REGION Network 3: Hardware Clock Memory 0.1S
   // 系统程序段 / System program segment
   RUNG wire#powerrail
      Contact( "Sys".COM.AlwaysON )
      wire#w1
      Contact( "ClockMemory0.1s" )
      Coil( "Sys".COM.FlashTime100mS )
   END_RUNG
   RUNG wire#w1
      Contact( "ClockMemory0.2s" )
      Coil( "Sys".COM.FlashTime200mS )
   END_RUNG
   RUNG wire#w1
      Contact( "ClockMemory0.5s" )
      Coil( "Sys".COM.FlashTime500mS )
   END_RUNG
   RUNG wire#w1
      Contact( "ClockMemory1s" )
      Coil( "Sys".COM.FlashTime1S )
   END_RUNG
   RUNG wire#w1
      Contact( "ClockMemory2s" )
      Coil( "Sys".COM.FlashTime2S )
   END_RUNG
   // the same network as SCL:
   "Sys".COM.FlashTime100mS := "Sys".COM.AlwaysON AND "ClockMemory0.1s";
   "Sys".COM.FlashTime200mS := "Sys".COM.AlwaysON AND "ClockMemory0.2s";
   "Sys".COM.FlashTime500mS := "Sys".COM.AlwaysON AND "ClockMemory0.5s";
   "Sys".COM.FlashTime1S := "Sys".COM.AlwaysON AND "ClockMemory1s";
   "Sys".COM.FlashTime2S := "Sys".COM.AlwaysON AND "ClockMemory2s";
END_REGION

REGION Network 4: Date and time config
   // 系统程序段 / System program segment
   RUNG wire#powerrail
      Contact( "Sys".DateTime.Trigger )
      { S7_Templates := "date_type := Date_And_Time" } WR_SYS_T(IN := "Sys".DateTime.Set, RET_VAL => "Sys".RETVALI)
      R_Coil( "Sys".DateTime.Trigger )
   END_RUNG
   // the same network as SCL:
   "Sys".RETVALI := WR_SYS_T(EN := "Sys".DateTime.Trigger, IN := "Sys".DateTime.Set, ENO => #_w1);
   IF #_w1 THEN "Sys".DateTime.Trigger := FALSE; END_IF;
END_REGION

REGION Network 5: Diagnostic
   RUNG wire#powerrail
      "Diagnostic"(iCPUType := 2, iDBNum := 3001, iOffset := 132, iHardwareID := "Local~PROFINET_IO-System", oStatus => "DiagnosticDataBlock".Profinet.PNReadStatus)
   END_RUNG
   // the same network as SCL:
   "Diagnostic"(iCPUType := 2,
                iDBNum := 3001,
                iOffset := 132,
                iHardwareID := "Local~PROFINET_IO-System",
                oStatus => "DiagnosticDataBlock".Profinet.PNReadStatus);
END_REGION

REGION Network 6 (SCL): Win
       "ST10_GeneralData".HMI.Win.WinBullfer := 0;
       FOR #i := 1 TO 10 DO
           "ST10_GeneralData".HMI.Win.WinBullfer := "ST10_GeneralData".HMI.Win.WinBullfer + "ST10_GeneralData".HMI.Win."10x弹窗"[#i] * 11 +"ST10_GeneralData".HMI.Win."20x弹窗"[2] * 21 +"ST10_GeneralData".HMI.Win."30x弹窗"[#i] * 31 +"ST10_GeneralData".HMI.Win."40x弹窗"[#i] * 41;
       END_FOR;
       "ST10_GeneralData".HMI.Win.WinBullfer := ABS("ST10_GeneralData".HMI.Win.WinBullfer);
       "ST10_GeneralData".HMI.Win.TON[1](IN := "ST10_GeneralData".HMI.Win.Win <> "ST10_GeneralData".HMI.Win.WinBullfer,
                          PT := T#0.5S);
   IF "ST10_GeneralData".HMI.Win.TON[1].Q THEN
       "ST10_GeneralData".HMI.Win.Win := "ST10_GeneralData".HMI.Win.WinBullfer;
       END_IF;
END_REGION

REGION Network 7: MES_Shopworx
END_REGION

REGION Network 8: Call Main
   // 系统程序段 / System program segment
   RUNG wire#powerrail
      "ST10_Main"()
   END_RUNG
   // the same network as SCL:
   "ST10_Main"();
END_REGION

REGION Network 9: DataHandling in HMI
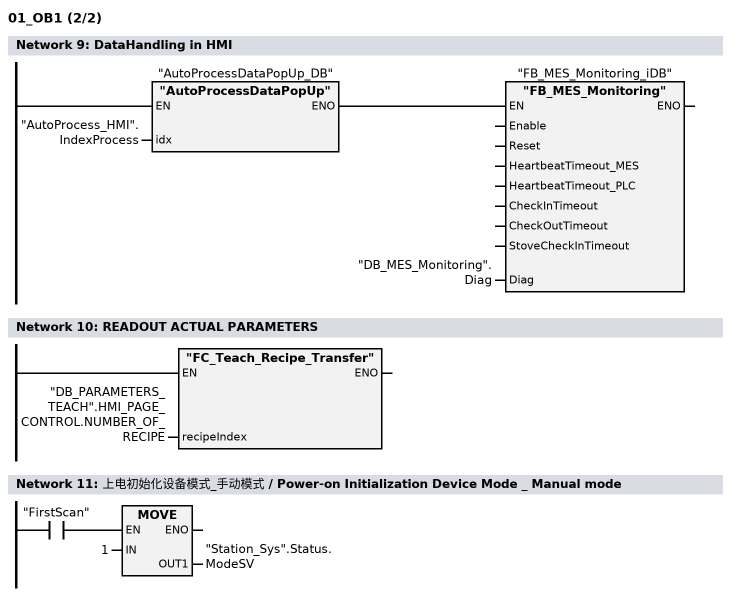
   RUNG wire#powerrail
      "AutoProcessDataPopUp_DB"(idx := "AutoProcess_HMI".IndexProcess)
      "FB_MES_Monitoring_iDB"(Enable :=, Reset :=, HeartbeatTimeout_MES :=, HeartbeatTimeout_PLC :=, CheckInTimeout :=, CheckOutTimeout :=, StoveCheckInTimeout :=, Diag := "DB_MES_Monitoring".Diag)
   END_RUNG
   // the same network as SCL:
   "AutoProcessDataPopUp_DB"(idx := "AutoProcess_HMI".IndexProcess, ENO => #_w1);   // "AutoProcessDataPopUp"
   IF #_w1 THEN
       "FB_MES_Monitoring_iDB"(Diag := "DB_MES_Monitoring".Diag);   // "FB_MES_Monitoring"
   END_IF;
END_REGION

REGION Network 10: READOUT ACTUAL PARAMETERS
   RUNG wire#powerrail
      "FC_Teach_Recipe_Transfer"(recipeIndex := "DB_PARAMETERS_TEACH".HMI_PAGE_CONTROL.NUMBER_OF_RECIPE)
   END_RUNG
   // the same network as SCL:
   "FC_Teach_Recipe_Transfer"(recipeIndex := "DB_PARAMETERS_TEACH".HMI_PAGE_CONTROL.NUMBER_OF_RECIPE);
END_REGION

REGION Network 11: 上电初始化设备模式_手动模式 / Power-on Initialization Device Mode _ Manual mode
   RUNG wire#powerrail
      Contact( "FirstScan" )
      Move(in := 1, out1 => "Station_Sys".Status.ModeSV)
   END_RUNG
   // the same network as SCL:
   IF "FirstScan" THEN "Station_Sys".Status.ModeSV := 1; END_IF;
END_REGION
END_ORGANIZATION_BLOCK

FUNCTION "Diagnostic" : Void   // FC3001, SCL
TITLE = Diagnostic
{ S7_Optimized_Access := 'FALSE' }
AUTHOR : STD
FAMILY : RCS
VERSION : 18.0
// stored: AutoNumber false, SetENOAutomatically true
   VAR_INPUT
      iCPUType : Int;   // 1-DP&PN 2-PN
      iDBNum : Word;
      iOffset : Int;   // Start address
      iHardwareID : HW_IOSYSTEM;
   END_VAR
   VAR_OUTPUT
      oStatus : Int;
   END_VAR
   VAR_TEMP
      RDSRet : Struct
         Busy : Bool;
         Header : Struct
            Length : Word;
            Number : Word;
         END_STRUCT;
      END_STRUCT;
      retInt : Int;
      SSL : Struct
         SSID : Word;
         Index : Word;
         Length : Int;
      END_STRUCT;
      DR : Any;
      DRS AT DR : Struct
         SyntaxID : Byte;
         DataType : Byte;
         RepetitionFactor : Int;
         DB_Number : Word;
         MemoryAreaAddress : DWord;
      END_STRUCT;
   END_VAR
BEGIN

   (*############################################################
      RUHLAMAT SUZHOU ELEC.STD.
      Copyright (c) 2017. All rights reserved.    

      NAME OF FUNCTION BLOCK:         Diagnostic
      VERSION NUMBER:                 V3.0
      COMPOSER:                       Ming.Jiang

      CreateDate:                    16.Nov.2016
      ----------------------------------------------------------
      Interface description:
      IN:
          "iCPUType"
          iDBNum
          iOffset
          iHardwareID

      INOUT:
      OUT:
          oStatus

      ----------------------------------------------------------
      #RET_VALUE:

      #Alert Value:

      ----------------------------------------------------------
      Date           Name      Version           Activity                                                                              
      28.Nov.2016    JM        V3.0              add alarm

   ############################################################*)
   IF #iCPUType = 0 OR #iDBNum = 0 THEN
       ENO := 0;
       RETURN;
   ELSE
       IF #iCPUType=2 THEN
           GOTO PN;
       ELSIF #iCPUType=1 THEN
           ;
       ELSE
           ENO := 0;
           RETURN;
       END_IF;
       #DRS.SyntaxID := 16#10;
       #DRS.DataType := 16#02;
       #DRS.RepetitionFactor := 128;
       #DRS.DB_Number := #iDBNum;
       #DRS.MemoryAreaAddress := 16#8400_0000 OR (SHL(IN := INT_TO_DWORD(#iOffset), N := 3));
       #oStatus := DeviceStates(LADDR := #iHardwareID, MODE := 2, STATE := #DR);
   PN:
       #DRS.SyntaxID := 16#10;
       #DRS.DataType := 16#02;
       #DRS.RepetitionFactor := 128;
       #DRS.DB_Number := #iDBNum;
       #DRS.MemoryAreaAddress := 16#8400_0000 OR (SHL(IN := INT_TO_DWORD(#iOffset), N := 3));
       #oStatus := DeviceStates(LADDR := #iHardwareID, MODE := 2, STATE := #DR);
       // orginise interface data 
       ENO := 1;
       RETURN;
   END_IF;
END_FUNCTION

FUNCTION "ST10_Main" : Void   // FC1050, LAD
{ S7_Optimized_Access := 'FALSE' }
// //=====================================================
// // INFO
// //=====================================================
// // NAME : ST10_Main
// // EN   : Main control logic for OP010 station.
// // ZH   : OP010 主控制逻辑。
// // SK   : Hlavná riadiaca logika stanice OP010.
// //=====================================================
// stored: AutoNumber false, SetENOAutomatically false
BEGIN

REGION Network 1 (SCL): INFO
   //=====================================================
   // INFO
   //=====================================================
   // NAME : ST10_Main
   // EN   : Main control logic for OP010 station.
   // ZH   : OP010 主控制逻辑。
   // SK   : Hlavná riadiaca logika stanice OP010.
   //=====================================================
END_REGION

REGION Network 2
   // 系统功能组调用部分
   // 1.该部分用户可以自己根据系统的组成将需要的功能块调用写在该部分
   // 2.该部分禁止与系统功能无关的程序在此处调用
END_REGION

NETWORK
TITLE = XXXX=====Station Relation/工位相关 =====StartXXXXX / XXXX=====Station Relation/Station correlation =====StartXXXXX

REGION Network 4: input /输入
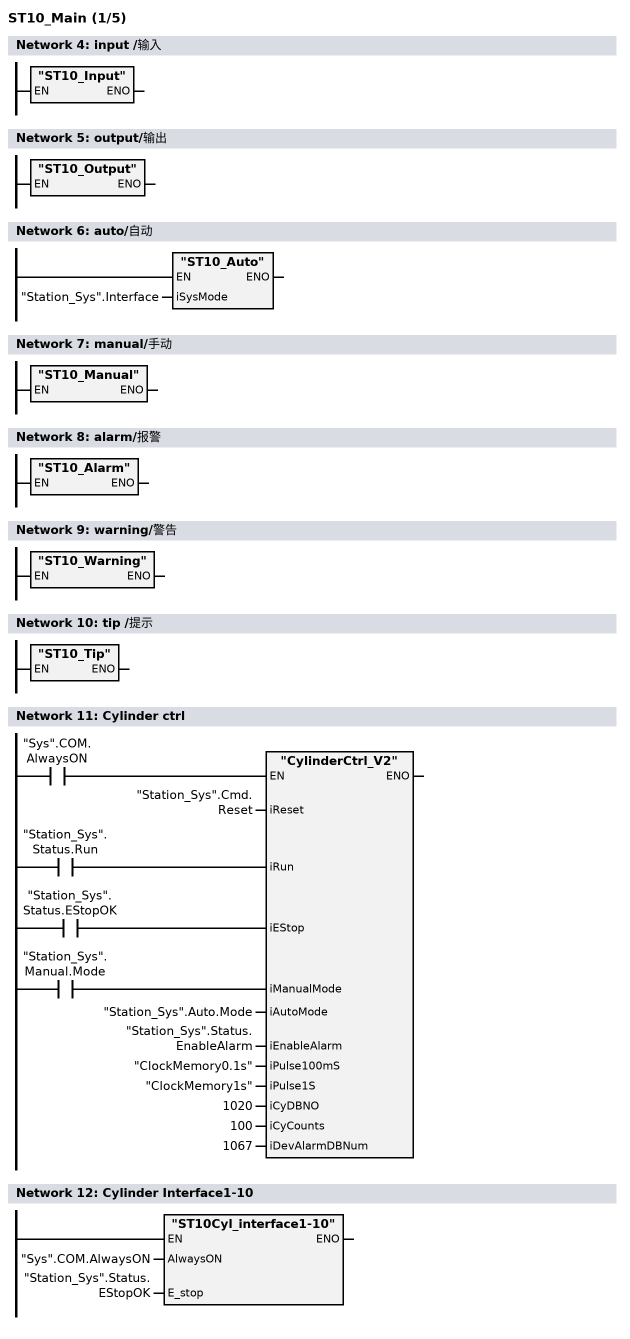
   RUNG wire#powerrail
      "ST10_Input"()
   END_RUNG
   // the same network as SCL:
   "ST10_Input"();
END_REGION

REGION Network 5: output/输出
   RUNG wire#powerrail
      "ST10_Output"()
   END_RUNG
   // the same network as SCL:
   "ST10_Output"();
END_REGION

REGION Network 6: auto/自动
   RUNG wire#powerrail
      "ST10_Auto"(iSysMode := "Station_Sys".Interface)
   END_RUNG
   // the same network as SCL:
   "ST10_Auto"(iSysMode := "Station_Sys".Interface);
END_REGION

REGION Network 7: manual/手动
   RUNG wire#powerrail
      "ST10_Manual"()
   END_RUNG
   // the same network as SCL:
   "ST10_Manual"();
END_REGION

REGION Network 8: alarm/报警
   RUNG wire#powerrail
      "ST10_Alarm"()
   END_RUNG
   // the same network as SCL:
   "ST10_Alarm"();
END_REGION

REGION Network 9: warning/警告
   RUNG wire#powerrail
      "ST10_Warning"()
   END_RUNG
   // the same network as SCL:
   "ST10_Warning"();
END_REGION

REGION Network 10: tip /提示
   RUNG wire#powerrail
      "ST10_Tip"()
   END_RUNG
   // the same network as SCL:
   "ST10_Tip"();
END_REGION

REGION Network 11: Cylinder ctrl
   RUNG wire#powerrail
      Contact( "Sys".COM.AlwaysON )
      "CylinderCtrl_V2"(iRun := wire#w1, iEStop := wire#w2, iManualMode := wire#w3, iReset := "Station_Sys".Cmd.Reset, iAutoMode := "Station_Sys".Auto.Mode, iEnableAlarm := "Station_Sys".Status.EnableAlarm, iPulse100mS := "ClockMemory0.1s", iPulse1S := "ClockMemory1s", iCyDBNO := 1020, iCyCounts := 100, iDevAlarmDBNum := 1067)
   END_RUNG
   RUNG wire#powerrail
      Contact( "Station_Sys".Status.Run )
   END_RUNG wire#w1
   RUNG wire#powerrail
      Contact( "Station_Sys".Status.EStopOK )
   END_RUNG wire#w2
   RUNG wire#powerrail
      Contact( "Station_Sys".Manual.Mode )
   END_RUNG wire#w3
   // the same network as SCL:
   IF "Sys".COM.AlwaysON THEN
       "CylinderCtrl_V2"(iReset := "Station_Sys".Cmd.Reset,
                         iRun := "Station_Sys".Status.Run,
                         iEStop := "Station_Sys".Status.EStopOK,
                         iManualMode := "Station_Sys".Manual.Mode,
                         iAutoMode := "Station_Sys".Auto.Mode,
                         iEnableAlarm := "Station_Sys".Status.EnableAlarm,
                         iPulse100mS := "ClockMemory0.1s",
                         iPulse1S := "ClockMemory1s",
                         iCyDBNO := 1020,
                         iCyCounts := 100,
                         iDevAlarmDBNum := 1067);
   END_IF;
END_REGION

REGION Network 12: Cylinder Interface1-10
   RUNG wire#powerrail
      "ST10Cyl_interface1-10"(AlwaysON := "Sys".COM.AlwaysON, E_stop := "Station_Sys".Status.EStopOK)
   END_RUNG
   // the same network as SCL:
   "ST10Cyl_interface1-10"(AlwaysON := "Sys".COM.AlwaysON, E_stop := "Station_Sys".Status.EStopOK);
END_REGION

REGION Network 13: Cylinder Interface11-20
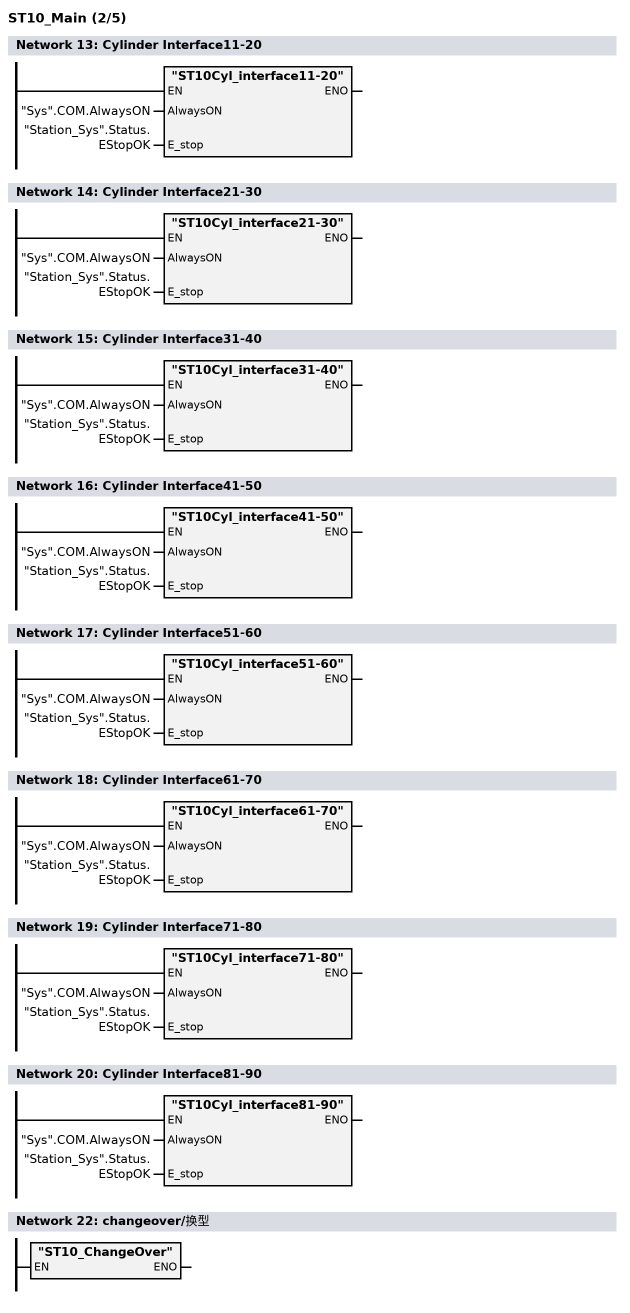
   RUNG wire#powerrail
      "ST10Cyl_interface11-20"(AlwaysON := "Sys".COM.AlwaysON, E_stop := "Station_Sys".Status.EStopOK)
   END_RUNG
   // the same network as SCL:
   "ST10Cyl_interface11-20"(AlwaysON := "Sys".COM.AlwaysON, E_stop := "Station_Sys".Status.EStopOK);
END_REGION

REGION Network 14: Cylinder Interface21-30
   RUNG wire#powerrail
      "ST10Cyl_interface21-30"(AlwaysON := "Sys".COM.AlwaysON, E_stop := "Station_Sys".Status.EStopOK)
   END_RUNG
   // the same network as SCL:
   "ST10Cyl_interface21-30"(AlwaysON := "Sys".COM.AlwaysON, E_stop := "Station_Sys".Status.EStopOK);
END_REGION

REGION Network 15: Cylinder Interface31-40
   RUNG wire#powerrail
      "ST10Cyl_interface31-40"(AlwaysON := "Sys".COM.AlwaysON, E_stop := "Station_Sys".Status.EStopOK)
   END_RUNG
   // the same network as SCL:
   "ST10Cyl_interface31-40"(AlwaysON := "Sys".COM.AlwaysON, E_stop := "Station_Sys".Status.EStopOK);
END_REGION

REGION Network 16: Cylinder Interface41-50
   RUNG wire#powerrail
      "ST10Cyl_interface41-50"(AlwaysON := "Sys".COM.AlwaysON, E_stop := "Station_Sys".Status.EStopOK)
   END_RUNG
   // the same network as SCL:
   "ST10Cyl_interface41-50"(AlwaysON := "Sys".COM.AlwaysON, E_stop := "Station_Sys".Status.EStopOK);
END_REGION

REGION Network 17: Cylinder Interface51-60
   RUNG wire#powerrail
      "ST10Cyl_interface51-60"(AlwaysON := "Sys".COM.AlwaysON, E_stop := "Station_Sys".Status.EStopOK)
   END_RUNG
   // the same network as SCL:
   "ST10Cyl_interface51-60"(AlwaysON := "Sys".COM.AlwaysON, E_stop := "Station_Sys".Status.EStopOK);
END_REGION

REGION Network 18: Cylinder Interface61-70
   RUNG wire#powerrail
      "ST10Cyl_interface61-70"(AlwaysON := "Sys".COM.AlwaysON, E_stop := "Station_Sys".Status.EStopOK)
   END_RUNG
   // the same network as SCL:
   "ST10Cyl_interface61-70"(AlwaysON := "Sys".COM.AlwaysON, E_stop := "Station_Sys".Status.EStopOK);
END_REGION

REGION Network 19: Cylinder Interface71-80
   RUNG wire#powerrail
      "ST10Cyl_interface71-80"(AlwaysON := "Sys".COM.AlwaysON, E_stop := "Station_Sys".Status.EStopOK)
   END_RUNG
   // the same network as SCL:
   "ST10Cyl_interface71-80"(AlwaysON := "Sys".COM.AlwaysON, E_stop := "Station_Sys".Status.EStopOK);
END_REGION

REGION Network 20: Cylinder Interface81-90
   RUNG wire#powerrail
      "ST10Cyl_interface81-90"(AlwaysON := "Sys".COM.AlwaysON, E_stop := "Station_Sys".Status.EStopOK)
   END_RUNG
   // the same network as SCL:
   "ST10Cyl_interface81-90"(AlwaysON := "Sys".COM.AlwaysON, E_stop := "Station_Sys".Status.EStopOK);
END_REGION

REGION Network 22: changeover/换型
   RUNG wire#powerrail
      "ST10_ChangeOver"()
   END_RUNG
   // the same network as SCL:
   "ST10_ChangeOver"();
END_REGION

REGION Network 23: Device
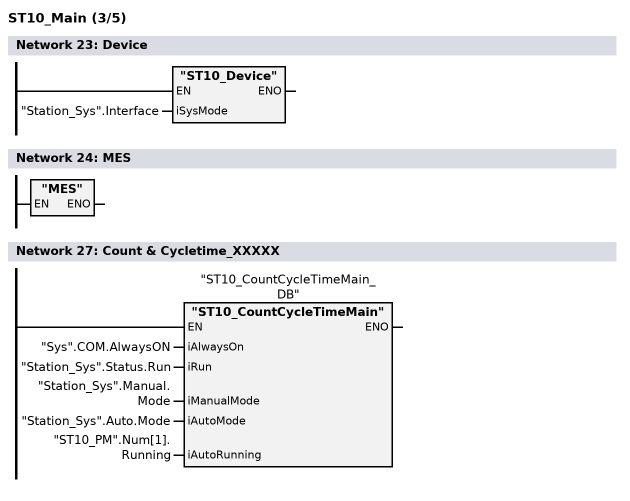
   RUNG wire#powerrail
      "ST10_Device"(iSysMode := "Station_Sys".Interface)
   END_RUNG
   // the same network as SCL:
   "ST10_Device"(iSysMode := "Station_Sys".Interface);
END_REGION

REGION Network 24: MES
   RUNG wire#powerrail
      "MES"()
   END_RUNG
   // the same network as SCL:
   "MES"();
END_REGION

REGION Network 25: =====System Function related information Section =====Start
END_REGION

NETWORK
TITLE = SystemFunction IO

REGION Network 27: Count & Cycletime_XXXXX
   RUNG wire#powerrail
      "ST10_CountCycleTimeMain_DB"(iAlwaysOn := "Sys".COM.AlwaysON, iRun := "Station_Sys".Status.Run, iManualMode := "Station_Sys".Manual.Mode, iAutoMode := "Station_Sys".Auto.Mode, iAutoRunning := "ST10_PM".Num[1].Running)
   END_RUNG
   // the same network as SCL:
   "ST10_CountCycleTimeMain_DB"(iAlwaysOn := "Sys".COM.AlwaysON,   // "ST10_CountCycleTimeMain"
                           iRun := "Station_Sys".Status.Run,
                           iManualMode := "Station_Sys".Manual.Mode,
                           iAutoMode := "Station_Sys".Auto.Mode,
                           iAutoRunning := "ST10_PM".Num[1].Running);
END_REGION

REGION Network 28: System mode
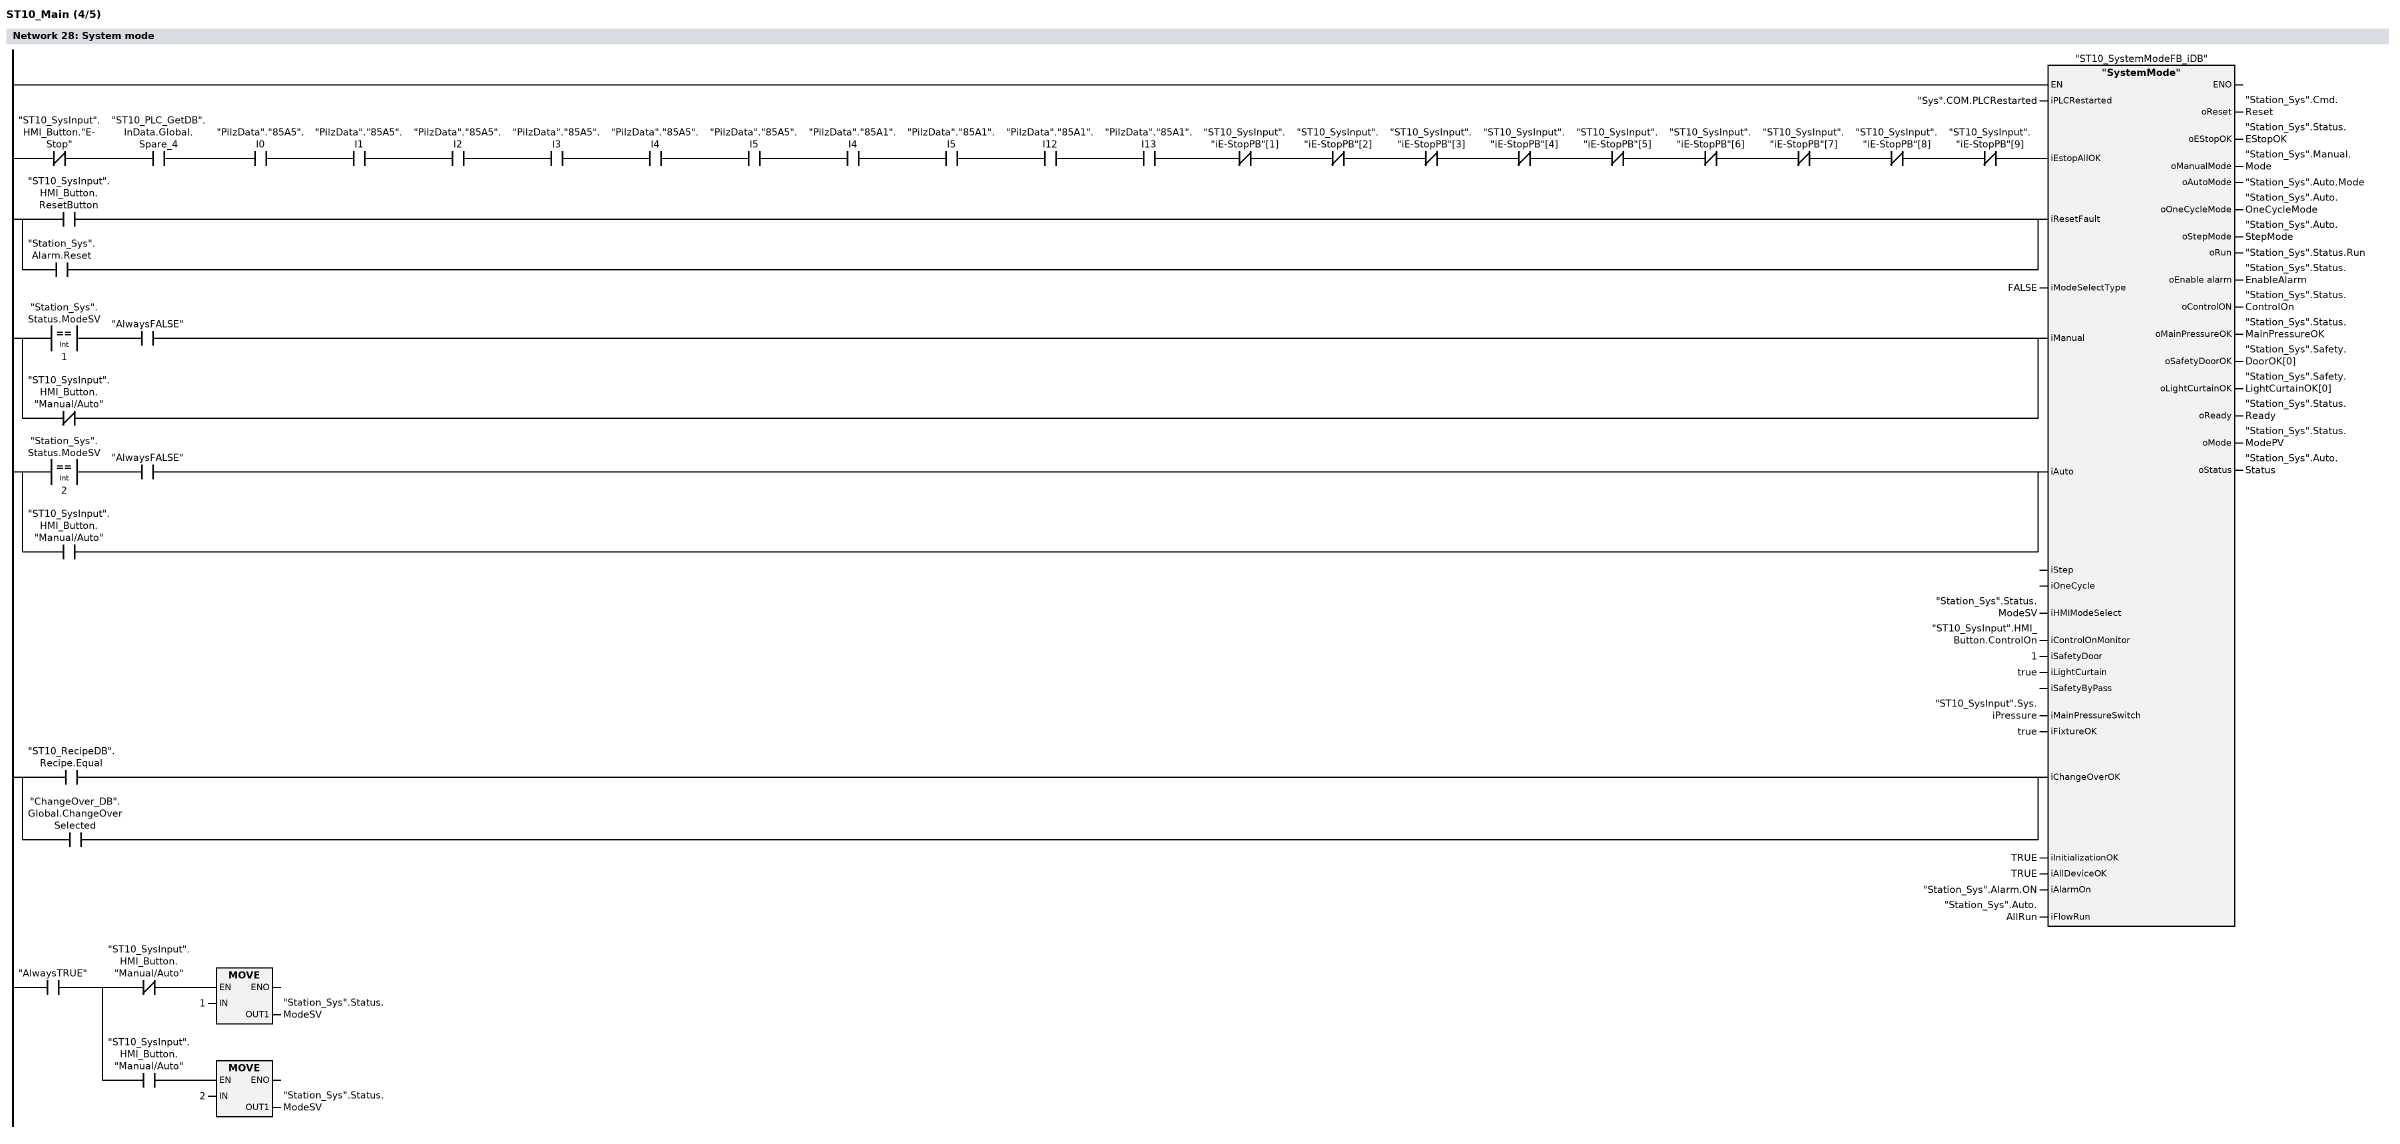
   RUNG wire#powerrail
      "ST10_SystemModeFB_iDB"(iEstopAllOK := wire#w1, iResetFault := wire#w2, iManual := wire#w3, iAuto := wire#w4, iChangeOverOK := wire#w5, iPLCRestarted := "Sys".COM.PLCRestarted, iModeSelectType := FALSE, iStep :=, iOneCycle :=, iHMIModeSelect := "Station_Sys".Status.ModeSV, iControlOnMonitor := "ST10_SysInput".HMI_Button.ControlOn, iSafetyDoor := 1, iLightCurtain := true, iSafetyByPass :=, iMainPressureSwitch := "ST10_SysInput".Sys.iPressure, iFixtureOK := true, iInitializationOK := TRUE, iAllDeviceOK := TRUE, iAlarmOn := "Station_Sys".Alarm.ON, iFlowRun := "Station_Sys".Auto.AllRun, oReset => "Station_Sys".Cmd.Reset, oEStopOK => "Station_Sys".Status.EStopOK, oManualMode => "Station_Sys".Manual.Mode, oAutoMode => "Station_Sys".Auto.Mode, oOneCycleMode => "Station_Sys".Auto.OneCycleMode, oStepMode => "Station_Sys".Auto.StepMode, oRun => "Station_Sys".Status.Run, "oEnable alarm" => "Station_Sys".Status.EnableAlarm, oControlON => "Station_Sys".Status.ControlOn, oMainPressureOK => "Station_Sys".Status.MainPressureOK, oSafetyDoorOK => "Station_Sys".Safety.DoorOK[0], oLightCurtainOK => "Station_Sys".Safety.LightCurtainOK[0], oReady => "Station_Sys".Status.Ready, oMode => "Station_Sys".Status.ModePV, oStatus => "Station_Sys".Auto.Status)
   END_RUNG
   RUNG wire#powerrail
      I_Contact( "ST10_SysInput".HMI_Button."E-Stop" )
      Contact( "ST10_PLC_GetDB".InData.Global.Spare_4 )
      Contact( "PilzData"."85A5".I0 )
      Contact( "PilzData"."85A5".I1 )
      Contact( "PilzData"."85A5".I2 )
      Contact( "PilzData"."85A5".I3 )
      Contact( "PilzData"."85A5".I4 )
      Contact( "PilzData"."85A5".I5 )
      Contact( "PilzData"."85A1".I4 )
      Contact( "PilzData"."85A1".I5 )
      Contact( "PilzData"."85A1".I12 )
      Contact( "PilzData"."85A1".I13 )
      I_Contact( "ST10_SysInput"."iE-StopPB"[1] )
      I_Contact( "ST10_SysInput"."iE-StopPB"[2] )
      I_Contact( "ST10_SysInput"."iE-StopPB"[3] )
      I_Contact( "ST10_SysInput"."iE-StopPB"[4] )
      I_Contact( "ST10_SysInput"."iE-StopPB"[5] )
      I_Contact( "ST10_SysInput"."iE-StopPB"[6] )
      I_Contact( "ST10_SysInput"."iE-StopPB"[7] )
      I_Contact( "ST10_SysInput"."iE-StopPB"[8] )
      I_Contact( "ST10_SysInput"."iE-StopPB"[9] )
   END_RUNG wire#w1
   RUNG wire#powerrail
      Contact( "ST10_SysInput".HMI_Button.ResetButton )
   END_RUNG wire#w2
   RUNG wire#powerrail
      Contact( "Station_Sys".Alarm.Reset )
   END_RUNG wire#w2
   RUNG wire#powerrail
      { S7_Templates := "SrcType := Int" } EQ_Contact(in1 := "Station_Sys".Status.ModeSV, in2 := 1)
      Contact( "AlwaysFALSE" )
   END_RUNG wire#w3
   RUNG wire#powerrail
      I_Contact( "ST10_SysInput".HMI_Button."Manual/Auto" )
   END_RUNG wire#w3
   RUNG wire#powerrail
      { S7_Templates := "SrcType := Int" } EQ_Contact(in1 := "Station_Sys".Status.ModeSV, in2 := 2)
      Contact( "AlwaysFALSE" )
   END_RUNG wire#w4
   RUNG wire#powerrail
      Contact( "ST10_SysInput".HMI_Button."Manual/Auto" )
   END_RUNG wire#w4
   RUNG wire#powerrail
      Contact( "ST10_RecipeDB".Recipe.Equal )
   END_RUNG wire#w5
   RUNG wire#powerrail
      Contact( "ChangeOver_DB".Global.ChangeOverSelected )
   END_RUNG wire#w5
   RUNG wire#powerrail
      Contact( "AlwaysTRUE" )
      wire#w6
      I_Contact( "ST10_SysInput".HMI_Button."Manual/Auto" )
      Move(in := 1, out1 => "Station_Sys".Status.ModeSV)
   END_RUNG
   RUNG wire#w6
      Contact( "ST10_SysInput".HMI_Button."Manual/Auto" )
      Move(in := 2, out1 => "Station_Sys".Status.ModeSV)
   END_RUNG
   // the same network as SCL:
   "ST10_SystemModeFB_iDB"(iPLCRestarted := "Sys".COM.PLCRestarted,   // "SystemMode"
                           iEstopAllOK := NOT "ST10_SysInput".HMI_Button."E-Stop" AND "ST10_PLC_GetDB".InData.Global.Spare_4 AND "PilzData"."85A5".I0 AND "PilzData"."85A5".I1 AND "PilzData"."85A5".I2 AND "PilzData"."85A5".I3 AND "PilzData"."85A5".I4 AND "PilzData"."85A5".I5 AND "PilzData"."85A1".I4 AND "PilzData"."85A1".I5 AND "PilzData"."85A1".I12 AND "PilzData"."85A1".I13 AND NOT "ST10_SysInput"."iE-StopPB"[1] AND NOT "ST10_SysInput"."iE-StopPB"[2] AND NOT "ST10_SysInput"."iE-StopPB"[3] AND NOT "ST10_SysInput"."iE-StopPB"[4] AND NOT "ST10_SysInput"."iE-StopPB"[5] AND NOT "ST10_SysInput"."iE-StopPB"[6] AND NOT "ST10_SysInput"."iE-StopPB"[7] AND NOT "ST10_SysInput"."iE-StopPB"[8] AND NOT "ST10_SysInput"."iE-StopPB"[9],
                           iResetFault := "ST10_SysInput".HMI_Button.ResetButton OR "Station_Sys".Alarm.Reset,
                           iModeSelectType := FALSE,
                           iManual := (("Station_Sys".Status.ModeSV = 1) AND "AlwaysFALSE") OR NOT "ST10_SysInput".HMI_Button."Manual/Auto",
                           iAuto := (("Station_Sys".Status.ModeSV = 2) AND "AlwaysFALSE") OR "ST10_SysInput".HMI_Button."Manual/Auto",
                           iHMIModeSelect := "Station_Sys".Status.ModeSV,
                           iControlOnMonitor := "ST10_SysInput".HMI_Button.ControlOn,
                           iSafetyDoor := 1,
                           iLightCurtain := true,
                           iMainPressureSwitch := "ST10_SysInput".Sys.iPressure,
                           iFixtureOK := true,
                           iChangeOverOK := "ST10_RecipeDB".Recipe.Equal OR "ChangeOver_DB".Global.ChangeOverSelected,
                           iInitializationOK := TRUE,
                           iAllDeviceOK := TRUE,
                           iAlarmOn := "Station_Sys".Alarm.ON,
                           iFlowRun := "Station_Sys".Auto.AllRun,
                           oReset => "Station_Sys".Cmd.Reset,
                           oEStopOK => "Station_Sys".Status.EStopOK,
                           oManualMode => "Station_Sys".Manual.Mode,
                           oAutoMode => "Station_Sys".Auto.Mode,
                           oOneCycleMode => "Station_Sys".Auto.OneCycleMode,
                           oStepMode => "Station_Sys".Auto.StepMode,
                           oRun => "Station_Sys".Status.Run,
                           "oEnable alarm" => "Station_Sys".Status.EnableAlarm,
                           oControlON => "Station_Sys".Status.ControlOn,
                           oMainPressureOK => "Station_Sys".Status.MainPressureOK,
                           oSafetyDoorOK => "Station_Sys".Safety.DoorOK[0],
                           oLightCurtainOK => "Station_Sys".Safety.LightCurtainOK[0],
                           oReady => "Station_Sys".Status.Ready,
                           oMode => "Station_Sys".Status.ModePV,
                           oStatus => "Station_Sys".Auto.Status);
   IF "AlwaysTRUE" AND NOT "ST10_SysInput".HMI_Button."Manual/Auto" THEN
       "Station_Sys".Status.ModeSV := 1;
   END_IF;
   IF "AlwaysTRUE" AND "ST10_SysInput".HMI_Button."Manual/Auto" THEN
       "Station_Sys".Status.ModeSV := 2;
   END_IF;
END_REGION

REGION Network 29: Start button
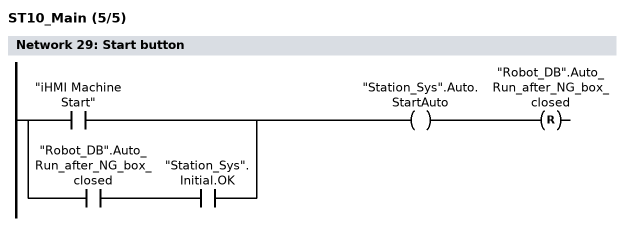
   RUNG wire#powerrail
      Contact( "iHMI Machine Start" )
      wire#w1
      Coil( "Station_Sys".Auto.StartAuto )
      R_Coil( "Robot_DB".Auto_Run_after_NG_box_closed )
   END_RUNG
   RUNG wire#powerrail
      Contact( "Robot_DB".Auto_Run_after_NG_box_closed )
      Contact( "Station_Sys".Initial.OK )
   END_RUNG wire#w1
   // the same network as SCL:
   "Station_Sys".Auto.StartAuto := "iHMI Machine Start" OR ("Robot_DB".Auto_Run_after_NG_box_closed AND "Station_Sys".Initial.OK);
   IF "Station_Sys".Auto.StartAuto THEN "Robot_DB".Auto_Run_after_NG_box_closed := FALSE; END_IF;
END_REGION

REGION Network 30 (SCL): System Interface
   "Station_Sys".Interface.CPUFristCycle  := "Sys".COM.PLCRestarted;
   "Station_Sys".Interface.SysRun         := "Station_Sys".Status.Run;
   "Station_Sys".Interface.Reset          := "Station_Sys".Cmd.Reset;
   "Station_Sys".Interface.EstopOK        := "Station_Sys".Status.EStopOK;
   "Station_Sys".Interface.SafetyDoorOK   := "Station_Sys".Safety.DoorOK[0];
   "Station_Sys".Interface.LightCurtainOK := "Station_Sys".Safety.LightCurtainOK[0];
   "Station_Sys".Interface.SetInitial     := "Station_Sys".Initial.Set;
   "Station_Sys".Interface.InitialRun     := "Station_Sys".Initial.Running;
   "Station_Sys".Interface.Ready          := "Station_Sys".Status.Ready;
   "Station_Sys".Interface.ManualMode     := "Station_Sys".Manual.Mode;
   "Station_Sys".Interface.Auto           := "Station_Sys".Auto;
END_REGION

REGION Network 31: =====System Function related information Section =====End
END_REGION

REGION Network 32: CallCalibration//标定调用
END_REGION

REGION Network 33 (SCL): ByPass Button
   // A
   "ST10_GeneralData".FunctionDeSelect.A.FunctionDeSelected_Servo380A1  := "ST10_GeneralData".FunctionDeSelect.A.DeSelectPB_Servo380A1;
   "ST10_GeneralData".FunctionDeSelect.A.FunctionDeSelected_Servo381A1  := "ST10_GeneralData".FunctionDeSelect.A.DeSelectPB_Servo381A1;
   "ST10_GeneralData".FunctionDeSelect.A.FunctionDeSelected_Servo383A1  := "ST10_GeneralData".FunctionDeSelect.A.DeSelectPB_Servo383A1;
   "ST10_GeneralData".FunctionDeSelect.A.FunctionDeSelected_Reader800A1 := "ST10_GeneralData".FunctionDeSelect.A.DeSelectPB_Reader800A1;
   "ST10_GeneralData".FunctionDeSelect.A.FunctionDeSelected_Reader801A1 := "ST10_GeneralData".FunctionDeSelect.A.DeSelectPB_Reader801A1;
   "ST10_GeneralData".FunctionDeSelect.A.FunctionDeSelected_Reader802A1 := "ST10_GeneralData".FunctionDeSelect.A.DeSelectPB_Reader802A1;
   "ST10_GeneralData".FunctionDeSelect.A.FunctionDeSelected_Reader803A1 := "ST10_GeneralData".FunctionDeSelect.A.DeSelectPB_Reader803A1;
   "ST10_GeneralData".FunctionDeSelect.A.FunctionDeSelected_Reader804A1 := "ST10_GeneralData".FunctionDeSelect.A.DeSelectPB_Reader804A1;

   // B
   "ST10_GeneralData".FunctionDeSelect.B.FunctionDeSelected_Press372A1     := "ST10_GeneralData".FunctionDeSelect.B.DeSelectPB_Press372A1;
   "ST10_GeneralData".FunctionDeSelect.B.FunctionDeSelected_Press375A1     := "ST10_GeneralData".FunctionDeSelect.B.DeSelectPB_Press375A1;
   "ST10_GeneralData".FunctionDeSelect.B.FunctionDeSelected_Reader806A1    := "ST10_GeneralData".FunctionDeSelect.B.DeSelectPB_Reader806A1;
   "ST10_GeneralData".FunctionDeSelect.B.FunctionDeSelected_TestPress372A1 := "ST10_GeneralData".FunctionDeSelect.B.DeSelectPB_TestPress372A1;
   "ST10_GeneralData".FunctionDeSelect.B.FunctionDeSelected_TestPress375A1 := "ST10_GeneralData".FunctionDeSelect.B.DeSelectPB_TestPress375A1;

   // C
   "ST10_GeneralData".FunctionDeSelect.C.FunctionDeSelected_Servo382A1 := "ST10_GeneralData".FunctionDeSelect.C.DeSelectPB_Servo382A1;
   "ST10_GeneralData".FunctionDeSelect.C.FunctionDeSelected_ServoIAI := "ST10_GeneralData".FunctionDeSelect.C.DeSelectPB_ServoIAI;
   "ST10_GeneralData".FunctionDeSelect.C.FunctionDeSelected_IV3810A1 := "ST10_GeneralData".FunctionDeSelect.C.DeSelectPB_IV3810A1;
   "ST10_GeneralData".FunctionDeSelect.C.FunctionDeSelected_IV3811A1 := "ST10_GeneralData".FunctionDeSelect.C.DeSelectPB_IV3811A1;
   "ST10_GeneralData".FunctionDeSelect.C.FunctionDeSelected_Glue := "ST10_GeneralData".FunctionDeSelect.C.DeSelectPB_Glue;

   // E
   "ST10_GeneralData".FunctionDeSelect.E.FunctionDeSelected := "ST10_GeneralData".FunctionDeSelect.E.DeSelectPB;

   // F
   "ST10_GeneralData".FunctionDeSelect.F.FunctionDeSelected_Reader805A1 := "ST10_GeneralData".FunctionDeSelect.F.DeSelectPB_Reader805A1;

   // H
   "ST10_GeneralData".FunctionDeSelect.H.FunctionDeSelected := "ST10_GeneralData".FunctionDeSelect.H.DeSelectPB;

   // J
   "ST10_GeneralData".FunctionDeSelect.J.FunctionDeSelected := "ST10_GeneralData".FunctionDeSelect.J.DeSelectPB;

   // K
   "ST10_GeneralData".FunctionDeSelect.K.FunctionDeSelected := "ST10_GeneralData".FunctionDeSelect.K.DeSelectPB;

   // L
   "ST10_GeneralData".FunctionDeSelect.L.FunctionDeSelected := "ST10_GeneralData".FunctionDeSelect.L.DeSelectPB;

   // MES
   "ST10_GeneralData".FunctionDeSelect.MES.FunctionDeSelected := "ST10_GeneralData".FunctionDeSelect.MES.DeSelectPB;

   //Auto>Maanual  ScanFixture
   "ST10_GeneralData".FunctionDeSelect.Global.FunctionDeSelected_ScanFixture := "ST10_GeneralData".FunctionDeSelect.Global.DeSelectPB_ScanFixture;
END_REGION
END_FUNCTION

FUNCTION "ST10_Input" : Void   // FC1001, LAD
{ S7_Optimized_Access := 'FALSE' }
VERSION : 0.1
// 注：本程序用来处理需要滤波，延时、计算的输入信号
// stored: AutoNumber false, IsIECCheckEnabled false, SetENOAutomatically false, UDAEnableTagReadback false
BEGIN

REGION Network 1 (SCL): HMI信号映射 / HMI signal mapping
   "ST10_SysInput".HMI_Button.ControlOn := "iHMI Control On";
   //"ST350_SysInput".HMI_Button.ControlOff:=
   "ST10_SysInput".HMI_Button.MachineStart := "iHMI Machine Start";
   "ST10_SysInput".HMI_Button.MachineStop := "iHMI Machine Stop";
   "ST10_SysInput".HMI_Button.ResetButton := "iHMI ResetButton";
   "ST10_SysInput".HMI_Button."Manual/Auto" := "iHMI Manual/Auto";
   "ST10_SysInput".HMI_Button.SafetyGateUnlock := "iHMI Safety Gate Unlock";
   "ST10_SysInput".HMI_Button."E-Stop" :=  "iHMI E-Stop";
END_REGION

REGION Network 2 (SCL): Sys IO Image
   "ST10_SysInput".Sys.iCircuitBreakerOK1 := "iCircuit Breaker OK_1";
   "ST10_SysInput".Sys.iCircuitBreakerOK2 := "iCircuit Breaker OK_2";
   "ST10_SysInput".Sys.iPressure:= "iPressure";
END_REGION

REGION Network 3 (SCL): iE-StopPB
   "ST10_SysInput"."iE-StopPB"[1] := "iE_StopButton2_A01";
   "ST10_SysInput"."iE-StopPB"[2] := "iE_StopButton3_A02";
   "ST10_SysInput"."iE-StopPB"[3] := "iE_StopButton4_H";
   "ST10_SysInput"."iE-StopPB"[4] := "iE_StopButton5_J";
   "ST10_SysInput"."iE-StopPB"[5] := "iE_StopButton6_K";
   "ST10_SysInput"."iE-StopPB"[6] := "iE_StopButton7_L";
   "ST10_SysInput"."iE-StopPB"[7] := "iH_StopButton";
   "ST10_SysInput"."iE-StopPB"[8] := "iJ_StopButton";
   "ST10_SysInput"."iE-StopPB"[9] := "iK_StopButton";
END_REGION

REGION Network 4 (SCL): iSafetyGatFeedBack
   (*
   "ST350_SysInput".iSafetyGatFeedBack[1] := "iSafety door Locking FeedBack_1";
   "ST350_SysInput".iSafetyGatFeedBack[2] := "iSafety door Locking FeedBack_2";
   "ST350_SysInput".iSafetyGatFeedBack[3] := "iSafety door Locking FeedBack_3";
   "ST350_SysInput".iSafetyGatFeedBack[4] := "iSafety door Locking FeedBack_4";
   "ST350_SysInput".iSafetyGatFeedBack[5] := "iSafety door Locking FeedBack_5";
   "ST350_SysInput".iSafetyGatFeedBack[6] := "iSafety door Locking FeedBack_6";
   "ST350_SysInput".iSafetyGatFeedBack[7] := "iSafety door Locking FeedBack_7";
   "ST350_SysInput".iSafetyGatFeedBack[8] := "iSafety door Locking FeedBack_8";
   *)
END_REGION

REGION Network 5 (SCL): iSafetydoorLockingFeedBack
   "ST10_SysInput".iSafetydoorLockingFeedBack[1] := "iSafety door Locking FeedBack_1";
   "ST10_SysInput".iSafetydoorLockingFeedBack[2] := "iSafety door Locking FeedBack_2";
   "ST10_SysInput".iSafetydoorLockingFeedBack[3] := "iSafety door Locking FeedBack_3";
   "ST10_SysInput".iSafetydoorLockingFeedBack[4] := "iSafety door Locking FeedBack_4";
   "ST10_SysInput".iSafetydoorLockingFeedBack[5] := "iSafety door Locking FeedBack_5";
   "ST10_SysInput".iSafetydoorLockingFeedBack[6] := "iSafety door Locking FeedBack_6";
   "ST10_SysInput".iSafetydoorLockingFeedBack[7] := "iSafety door Locking FeedBack_7";
   "ST10_SysInput".iSafetydoorLockingFeedBack[8] := "iSafety door Locking FeedBack_8";
END_REGION

REGION Network 6 (SCL): iSafetydoorLockingFeedBack
   "ST10_SysInput".iMaterieldoorLockingFeedBack[1] := "iMateriel Door Locking FeedBack_H1";
   "ST10_SysInput".iMaterieldoorLockingFeedBack[2] := "iMateriel Door Locking FeedBack_H2";
   "ST10_SysInput".iMaterieldoorLockingFeedBack[3] := "iMateriel Door Locking FeedBack_J1";
   "ST10_SysInput".iMaterieldoorLockingFeedBack[4] := "iMateriel Door Locking FeedBack_J2";
   "ST10_SysInput".iMaterieldoorLockingFeedBack[5] := "iMateriel Door Locking FeedBack_K1";
   "ST10_SysInput".iMaterieldoorLockingFeedBack[6] := "iMateriel Door Locking FeedBack_K2";
   "ST10_SysInput".iMaterieldoorLockingFeedBack[7] := "iMateriel Door Locking FeedBack_L1";
END_REGION
END_FUNCTION

FUNCTION "ST10_Output" : Void   // FC1002, LAD
{ S7_Optimized_Access := 'FALSE' }
// stored: AutoNumber false, SetENOAutomatically false
   VAR_TEMP   // added for the SCL form of the ladder/FBD networks
      _w1 : Bool;
      _w2 : Bool;
      _w3 : Bool;
      _w4 : Bool;
      _w5 : Bool;
      _w6 : Bool;
   END_VAR
BEGIN

REGION Network 1 (SCL): 安全门锁定信号映射SafetyDoorCoil / Security door lock_1
   "oSafetyDoorLocked_1" := "ST10_SysOutput".SafetyDoorCoil[1];
   "oSafetyDoorLocked_2" := "ST10_SysOutput".SafetyDoorCoil[2];
   "oSafetyDoorLocked_3" := "ST10_SysOutput".SafetyDoorCoil[3];
   "oSafetyDoorLocked_4" := "ST10_SysOutput".SafetyDoorCoil[4];
   "oSafetyDoorLocked_5" := "ST10_SysOutput".SafetyDoorCoil[5];
   "oSafetyDoorLocked_6" := "ST10_SysOutput".SafetyDoorCoil[6];
   "oSafetyDoorLocked_7" := "ST10_SysOutput".SafetyDoorCoil[7];
   "oSafetyDoorLocked_8" := "ST10_SysOutput".SafetyDoorCoil[8];
   "oSafetyDoorLocked" := "ST10_SysOutput".SafetyDoorCoil[9];
END_REGION

REGION Network 2 (SCL): 安全门锁定信号映射SafetyDoorCoil / Material door lock_1
   "oMaterielDoorLocked_H1" := "ST10_SysOutput".MaterialDoorCoil[1];
   "oMaterielDoorLocked_H2" := "ST10_SysOutput".MaterialDoorCoil[2];
   "oMaterielDoorLocked_J1" := "ST10_SysOutput".MaterialDoorCoil[3];
   "oMaterielDoorLocked_J2" := "ST10_SysOutput".MaterialDoorCoil[4];
   "oMaterielDoorLocked_K1" := "ST10_SysOutput".MaterialDoorCoil[5];
   "oMaterielDoorLocked_K2" := "ST10_SysOutput".MaterialDoorCoil[6];
   "oMaterielDoorLocked_L1" := "ST10_SysOutput".MaterialDoorCoil[7];


   "oE-NG-01SafetyGate" := "ST10_SysOutput".MaterialDoorCoil[8];
   "oE-NG-02SafetyGate" := "ST10_SysOutput".MaterialDoorCoil[9];
END_REGION

REGION Network 3: 塔灯
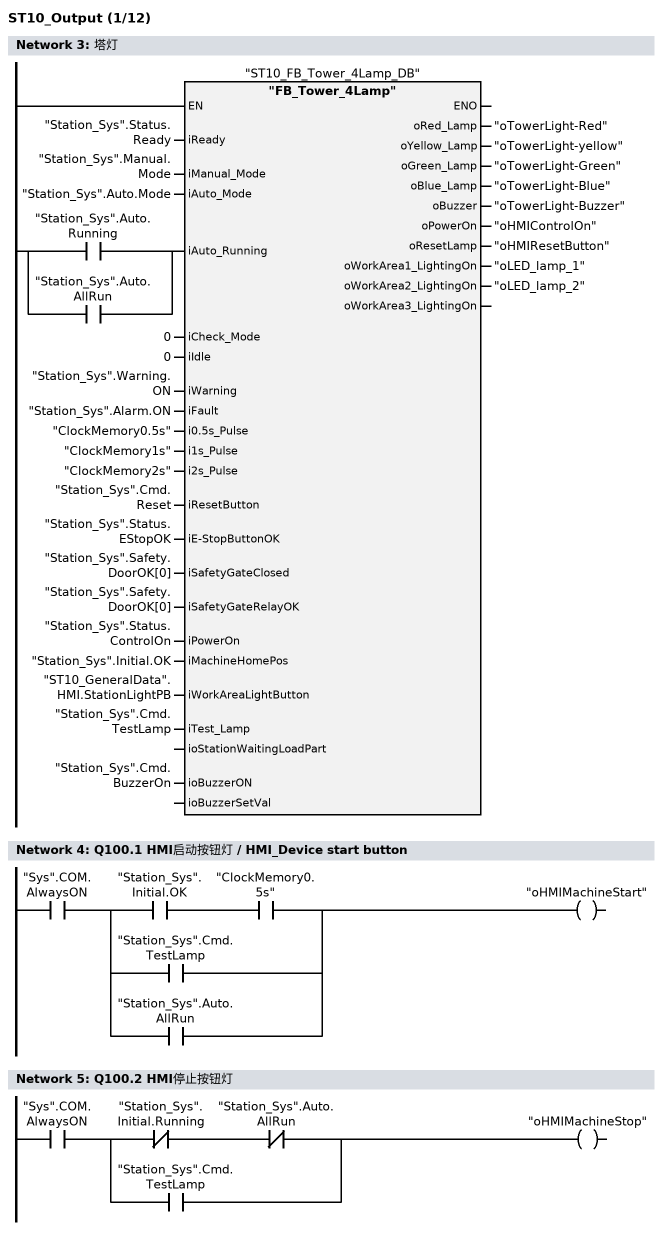
   RUNG wire#powerrail
      "ST10_FB_Tower_4Lamp_DB"(iAuto_Running := wire#w1, iReady := "Station_Sys".Status.Ready, iManual_Mode := "Station_Sys".Manual.Mode, iAuto_Mode := "Station_Sys".Auto.Mode, iCheck_Mode := 0, iIdle := 0, iWarning := "Station_Sys".Warning.ON, iFault := "Station_Sys".Alarm.ON, "i0.5s_Pulse" := "ClockMemory0.5s", i1s_Pulse := "ClockMemory1s", i2s_Pulse := "ClockMemory2s", iResetButton := "Station_Sys".Cmd.Reset, "iE-StopButtonOK" := "Station_Sys".Status.EStopOK, iSafetyGateClosed := "Station_Sys".Safety.DoorOK[0], iSafetyGateRelayOK := "Station_Sys".Safety.DoorOK[0], iPowerOn := "Station_Sys".Status.ControlOn, iMachineHomePos := "Station_Sys".Initial.OK, iWorkAreaLightButton := "ST10_GeneralData".HMI.StationLightPB, iTest_Lamp := "Station_Sys".Cmd.TestLamp, ioStationWaitingLoadPart :=, ioBuzzerON := "Station_Sys".Cmd.BuzzerOn, ioBuzzerSetVal :=, oRed_Lamp => "oTowerLight-Red", oYellow_Lamp => "oTowerLight-yellow", oGreen_Lamp => "oTowerLight-Green", oBlue_Lamp => "oTowerLight-Blue", oBuzzer => "oTowerLight-Buzzer", oPowerOn => "oHMIControlOn", oResetLamp => "oHMIResetButton", oWorkArea1_LightingOn => "oLED_lamp_1", oWorkArea2_LightingOn => "oLED_lamp_2", oWorkArea3_LightingOn =>)
   END_RUNG
   RUNG wire#powerrail
      Contact( "Station_Sys".Auto.Running )
   END_RUNG wire#w1
   RUNG wire#powerrail
      Contact( "Station_Sys".Auto.AllRun )
   END_RUNG wire#w1
   // the same network as SCL:
   "ST10_FB_Tower_4Lamp_DB"(iReady := "Station_Sys".Status.Ready,   // "FB_Tower_4Lamp"
                           iManual_Mode := "Station_Sys".Manual.Mode,
                           iAuto_Mode := "Station_Sys".Auto.Mode,
                           iAuto_Running := "Station_Sys".Auto.Running OR "Station_Sys".Auto.AllRun,
                           iCheck_Mode := 0,
                           iIdle := 0,
                           iWarning := "Station_Sys".Warning.ON,
                           iFault := "Station_Sys".Alarm.ON,
                           "i0.5s_Pulse" := "ClockMemory0.5s",
                           i1s_Pulse := "ClockMemory1s",
                           i2s_Pulse := "ClockMemory2s",
                           iResetButton := "Station_Sys".Cmd.Reset,
                           "iE-StopButtonOK" := "Station_Sys".Status.EStopOK,
                           iSafetyGateClosed := "Station_Sys".Safety.DoorOK[0],
                           iSafetyGateRelayOK := "Station_Sys".Safety.DoorOK[0],
                           iPowerOn := "Station_Sys".Status.ControlOn,
                           iMachineHomePos := "Station_Sys".Initial.OK,
                           iWorkAreaLightButton := "ST10_GeneralData".HMI.StationLightPB,
                           iTest_Lamp := "Station_Sys".Cmd.TestLamp,
                           ioBuzzerON := "Station_Sys".Cmd.BuzzerOn,
                           oRed_Lamp => "oTowerLight-Red",
                           oYellow_Lamp => "oTowerLight-yellow",
                           oGreen_Lamp => "oTowerLight-Green",
                           oBlue_Lamp => "oTowerLight-Blue",
                           oBuzzer => "oTowerLight-Buzzer",
                           oPowerOn => "oHMIControlOn",
                           oResetLamp => "oHMIResetButton",
                           oWorkArea1_LightingOn => "oLED_lamp_1",
                           oWorkArea2_LightingOn => "oLED_lamp_2");
END_REGION

REGION Network 4: Q100.1 HMI启动按钮灯 / HMI_Device start button
   RUNG wire#powerrail
      Contact( "Sys".COM.AlwaysON )
      wire#w1
      Contact( "Station_Sys".Initial.OK )
      Contact( "ClockMemory0.5s" )
      wire#w2
      Coil( "oHMIMachineStart" )
   END_RUNG
   RUNG wire#w1
      Contact( "Station_Sys".Cmd.TestLamp )
   END_RUNG wire#w2
   RUNG wire#w1
      Contact( "Station_Sys".Auto.AllRun )
   END_RUNG wire#w2
   // the same network as SCL:
   "oHMIMachineStart" := "Sys".COM.AlwaysON AND (("Station_Sys".Initial.OK AND "ClockMemory0.5s") OR "Station_Sys".Cmd.TestLamp OR "Station_Sys".Auto.AllRun);
END_REGION

REGION Network 5: Q100.2 HMI停止按钮灯
   RUNG wire#powerrail
      Contact( "Sys".COM.AlwaysON )
      wire#w1
      I_Contact( "Station_Sys".Initial.Running )
      I_Contact( "Station_Sys".Auto.AllRun )
      wire#w2
      Coil( "oHMIMachineStop" )
   END_RUNG
   RUNG wire#w1
      Contact( "Station_Sys".Cmd.TestLamp )
   END_RUNG wire#w2
   // the same network as SCL:
   "oHMIMachineStop" := "Sys".COM.AlwaysON AND ((NOT "Station_Sys".Initial.Running AND NOT "Station_Sys".Auto.AllRun) OR "Station_Sys".Cmd.TestLamp);
END_REGION

REGION Network 6: Q100.4 HMI开门按钮灯
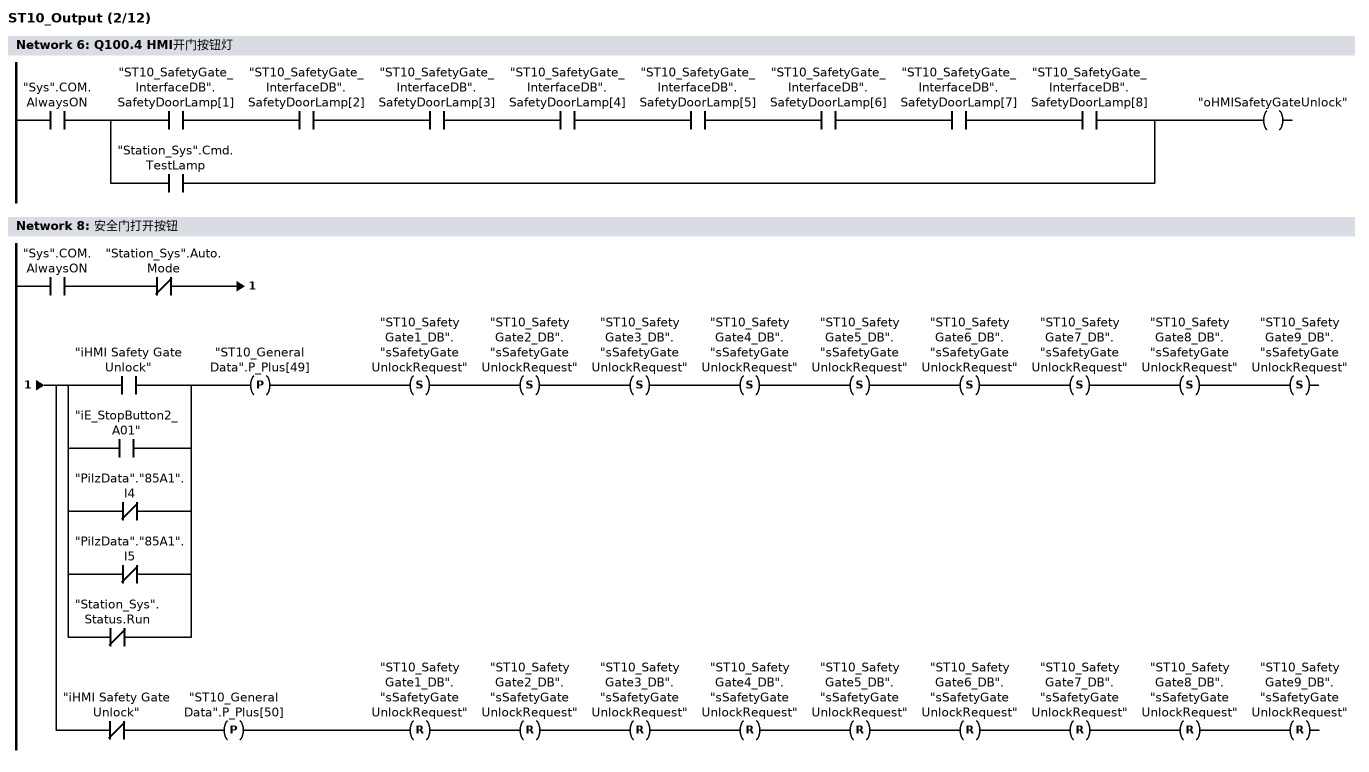
   RUNG wire#powerrail
      Contact( "Sys".COM.AlwaysON )
      wire#w1
      Contact( "ST10_SafetyGate_InterfaceDB".SafetyDoorLamp[1] )
      Contact( "ST10_SafetyGate_InterfaceDB".SafetyDoorLamp[2] )
      Contact( "ST10_SafetyGate_InterfaceDB".SafetyDoorLamp[3] )
      Contact( "ST10_SafetyGate_InterfaceDB".SafetyDoorLamp[4] )
      Contact( "ST10_SafetyGate_InterfaceDB".SafetyDoorLamp[5] )
      Contact( "ST10_SafetyGate_InterfaceDB".SafetyDoorLamp[6] )
      Contact( "ST10_SafetyGate_InterfaceDB".SafetyDoorLamp[7] )
      Contact( "ST10_SafetyGate_InterfaceDB".SafetyDoorLamp[8] )
      wire#w2
      Coil( "oHMISafetyGateUnlock" )
   END_RUNG
   RUNG wire#w1
      Contact( "Station_Sys".Cmd.TestLamp )
   END_RUNG wire#w2
   // the same network as SCL:
   "oHMISafetyGateUnlock" := "Sys".COM.AlwaysON AND (("ST10_SafetyGate_InterfaceDB".SafetyDoorLamp[1] AND "ST10_SafetyGate_InterfaceDB".SafetyDoorLamp[2] AND "ST10_SafetyGate_InterfaceDB".SafetyDoorLamp[3] AND "ST10_SafetyGate_InterfaceDB".SafetyDoorLamp[4] AND "ST10_SafetyGate_InterfaceDB".SafetyDoorLamp[5] AND "ST10_SafetyGate_InterfaceDB".SafetyDoorLamp[6] AND "ST10_SafetyGate_InterfaceDB".SafetyDoorLamp[7] AND "ST10_SafetyGate_InterfaceDB".SafetyDoorLamp[8]) OR "Station_Sys".Cmd.TestLamp);
END_REGION

REGION Network 8: 安全门打开按钮
   RUNG wire#powerrail
      Contact( "Sys".COM.AlwaysON )
      I_Contact( "Station_Sys".Auto.Mode )
      wire#w1
      Contact( "iHMI Safety Gate Unlock" )
      wire#w2
      P_Trig( "ST10_GeneralData".P_Plus[49] )
      S_Coil( "ST10_SafetyGate1_DB"."sSafetyGate UnlockRequest" )
      S_Coil( "ST10_SafetyGate2_DB"."sSafetyGate UnlockRequest" )
      S_Coil( "ST10_SafetyGate3_DB"."sSafetyGate UnlockRequest" )
      S_Coil( "ST10_SafetyGate4_DB"."sSafetyGate UnlockRequest" )
      S_Coil( "ST10_SafetyGate5_DB"."sSafetyGate UnlockRequest" )
      S_Coil( "ST10_SafetyGate6_DB"."sSafetyGate UnlockRequest" )
      S_Coil( "ST10_SafetyGate7_DB"."sSafetyGate UnlockRequest" )
      S_Coil( "ST10_SafetyGate8_DB"."sSafetyGate UnlockRequest" )
      S_Coil( "ST10_SafetyGate9_DB"."sSafetyGate UnlockRequest" )
   END_RUNG
   RUNG wire#w1
      Contact( "iE_StopButton2_A01" )
   END_RUNG wire#w2
   RUNG wire#w1
      I_Contact( "PilzData"."85A1".I4 )
   END_RUNG wire#w2
   RUNG wire#w1
      I_Contact( "PilzData"."85A1".I5 )
   END_RUNG wire#w2
   RUNG wire#w1
      I_Contact( "Station_Sys".Status.Run )
   END_RUNG wire#w2
   RUNG wire#w1
      I_Contact( "iHMI Safety Gate Unlock" )
      P_Trig( "ST10_GeneralData".P_Plus[50] )
      R_Coil( "ST10_SafetyGate1_DB"."sSafetyGate UnlockRequest" )
      R_Coil( "ST10_SafetyGate2_DB"."sSafetyGate UnlockRequest" )
      R_Coil( "ST10_SafetyGate3_DB"."sSafetyGate UnlockRequest" )
      R_Coil( "ST10_SafetyGate4_DB"."sSafetyGate UnlockRequest" )
      R_Coil( "ST10_SafetyGate5_DB"."sSafetyGate UnlockRequest" )
      R_Coil( "ST10_SafetyGate6_DB"."sSafetyGate UnlockRequest" )
      R_Coil( "ST10_SafetyGate7_DB"."sSafetyGate UnlockRequest" )
      R_Coil( "ST10_SafetyGate8_DB"."sSafetyGate UnlockRequest" )
      R_Coil( "ST10_SafetyGate9_DB"."sSafetyGate UnlockRequest" )
   END_RUNG
   // the same network as SCL:
   #_w1 := "Sys".COM.AlwaysON AND NOT "Station_Sys".Auto.Mode;
   #_w2 := #_w1 AND ("iHMI Safety Gate Unlock" OR "iE_StopButton2_A01" OR NOT "PilzData"."85A1".I4 OR NOT "PilzData"."85A1".I5 OR NOT "Station_Sys".Status.Run);
   #_w3 := #_w2 AND NOT "ST10_GeneralData".P_Plus[49];   // rising edge
   "ST10_GeneralData".P_Plus[49] := #_w2;
   IF #_w3 THEN
       "ST10_SafetyGate1_DB"."sSafetyGate UnlockRequest" := TRUE;
       "ST10_SafetyGate2_DB"."sSafetyGate UnlockRequest" := TRUE;
       "ST10_SafetyGate3_DB"."sSafetyGate UnlockRequest" := TRUE;
       "ST10_SafetyGate4_DB"."sSafetyGate UnlockRequest" := TRUE;
       "ST10_SafetyGate5_DB"."sSafetyGate UnlockRequest" := TRUE;
       "ST10_SafetyGate6_DB"."sSafetyGate UnlockRequest" := TRUE;
       "ST10_SafetyGate7_DB"."sSafetyGate UnlockRequest" := TRUE;
       "ST10_SafetyGate8_DB"."sSafetyGate UnlockRequest" := TRUE;
       "ST10_SafetyGate9_DB"."sSafetyGate UnlockRequest" := TRUE;
   END_IF;
   #_w4 := #_w1 AND NOT "iHMI Safety Gate Unlock";
   #_w5 := #_w4 AND NOT "ST10_GeneralData".P_Plus[50];   // rising edge
   "ST10_GeneralData".P_Plus[50] := #_w4;
   IF #_w5 THEN
       "ST10_SafetyGate1_DB"."sSafetyGate UnlockRequest" := FALSE;
       "ST10_SafetyGate2_DB"."sSafetyGate UnlockRequest" := FALSE;
       "ST10_SafetyGate3_DB"."sSafetyGate UnlockRequest" := FALSE;
       "ST10_SafetyGate4_DB"."sSafetyGate UnlockRequest" := FALSE;
       "ST10_SafetyGate5_DB"."sSafetyGate UnlockRequest" := FALSE;
       "ST10_SafetyGate6_DB"."sSafetyGate UnlockRequest" := FALSE;
       "ST10_SafetyGate7_DB"."sSafetyGate UnlockRequest" := FALSE;
       "ST10_SafetyGate8_DB"."sSafetyGate UnlockRequest" := FALSE;
       "ST10_SafetyGate9_DB"."sSafetyGate UnlockRequest" := FALSE;
   END_IF;
END_REGION

REGION Network 9: 安全门关闭
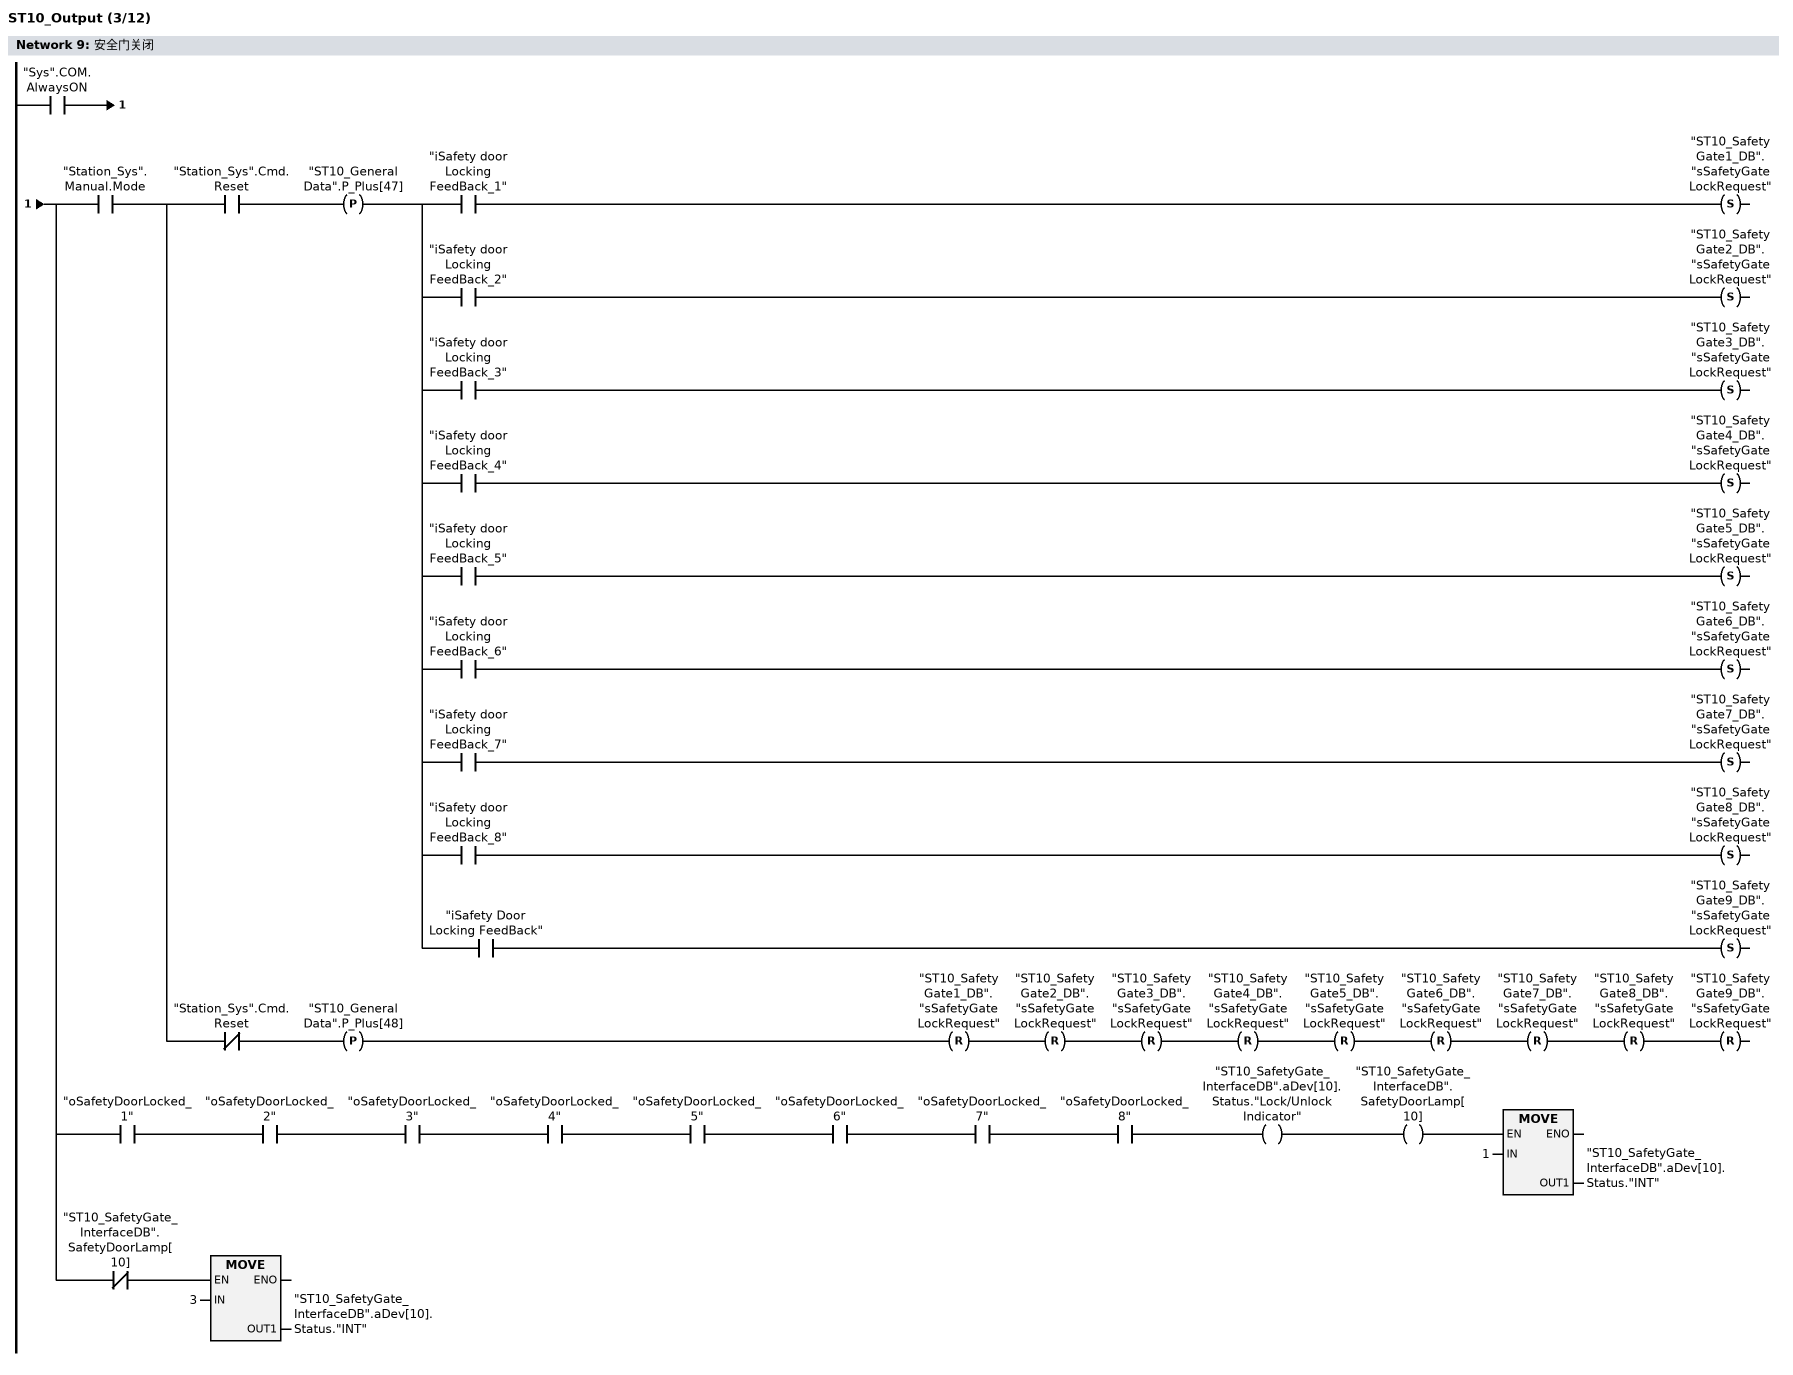
   RUNG wire#powerrail
      Contact( "Sys".COM.AlwaysON )
      wire#w1
      Contact( "Station_Sys".Manual.Mode )
      wire#w2
      Contact( "Station_Sys".Cmd.Reset )
      P_Trig( "ST10_GeneralData".P_Plus[47] )
      wire#w3
      Contact( "iSafety door Locking FeedBack_1" )
      S_Coil( "ST10_SafetyGate1_DB"."sSafetyGate LockRequest" )
   END_RUNG
   RUNG wire#w3
      Contact( "iSafety door Locking FeedBack_2" )
      S_Coil( "ST10_SafetyGate2_DB"."sSafetyGate LockRequest" )
   END_RUNG
   RUNG wire#w3
      Contact( "iSafety door Locking FeedBack_3" )
      S_Coil( "ST10_SafetyGate3_DB"."sSafetyGate LockRequest" )
   END_RUNG
   RUNG wire#w3
      Contact( "iSafety door Locking FeedBack_4" )
      S_Coil( "ST10_SafetyGate4_DB"."sSafetyGate LockRequest" )
   END_RUNG
   RUNG wire#w3
      Contact( "iSafety door Locking FeedBack_5" )
      S_Coil( "ST10_SafetyGate5_DB"."sSafetyGate LockRequest" )
   END_RUNG
   RUNG wire#w3
      Contact( "iSafety door Locking FeedBack_6" )
      S_Coil( "ST10_SafetyGate6_DB"."sSafetyGate LockRequest" )
   END_RUNG
   RUNG wire#w3
      Contact( "iSafety door Locking FeedBack_7" )
      S_Coil( "ST10_SafetyGate7_DB"."sSafetyGate LockRequest" )
   END_RUNG
   RUNG wire#w3
      Contact( "iSafety door Locking FeedBack_8" )
      S_Coil( "ST10_SafetyGate8_DB"."sSafetyGate LockRequest" )
   END_RUNG
   RUNG wire#w3
      Contact( "iSafety Door Locking FeedBack" )
      S_Coil( "ST10_SafetyGate9_DB"."sSafetyGate LockRequest" )
   END_RUNG
   RUNG wire#w2
      I_Contact( "Station_Sys".Cmd.Reset )
      P_Trig( "ST10_GeneralData".P_Plus[48] )
      R_Coil( "ST10_SafetyGate1_DB"."sSafetyGate LockRequest" )
      R_Coil( "ST10_SafetyGate2_DB"."sSafetyGate LockRequest" )
      R_Coil( "ST10_SafetyGate3_DB"."sSafetyGate LockRequest" )
      R_Coil( "ST10_SafetyGate4_DB"."sSafetyGate LockRequest" )
      R_Coil( "ST10_SafetyGate5_DB"."sSafetyGate LockRequest" )
      R_Coil( "ST10_SafetyGate6_DB"."sSafetyGate LockRequest" )
      R_Coil( "ST10_SafetyGate7_DB"."sSafetyGate LockRequest" )
      R_Coil( "ST10_SafetyGate8_DB"."sSafetyGate LockRequest" )
      R_Coil( "ST10_SafetyGate9_DB"."sSafetyGate LockRequest" )
   END_RUNG
   RUNG wire#w1
      Contact( "oSafetyDoorLocked_1" )
      Contact( "oSafetyDoorLocked_2" )
      Contact( "oSafetyDoorLocked_3" )
      Contact( "oSafetyDoorLocked_4" )
      Contact( "oSafetyDoorLocked_5" )
      Contact( "oSafetyDoorLocked_6" )
      Contact( "oSafetyDoorLocked_7" )
      Contact( "oSafetyDoorLocked_8" )
      Coil( "ST10_SafetyGate_InterfaceDB".aDev[10].Status."Lock/Unlock Indicator" )
      Coil( "ST10_SafetyGate_InterfaceDB".SafetyDoorLamp[10] )
      Move(in := 1, out1 => "ST10_SafetyGate_InterfaceDB".aDev[10].Status."INT")
   END_RUNG
   RUNG wire#w1
      I_Contact( "ST10_SafetyGate_InterfaceDB".SafetyDoorLamp[10] )
      Move(in := 3, out1 => "ST10_SafetyGate_InterfaceDB".aDev[10].Status."INT")
   END_RUNG
   // the same network as SCL:
   #_w1 := "Sys".COM.AlwaysON AND "Station_Sys".Manual.Mode;
   #_w2 := #_w1 AND "Station_Sys".Cmd.Reset;
   #_w3 := #_w2 AND NOT "ST10_GeneralData".P_Plus[47];   // rising edge
   "ST10_GeneralData".P_Plus[47] := #_w2;
   IF #_w3 AND "iSafety door Locking FeedBack_1" THEN
       "ST10_SafetyGate1_DB"."sSafetyGate LockRequest" := TRUE;
   END_IF;
   IF #_w3 AND "iSafety door Locking FeedBack_2" THEN
       "ST10_SafetyGate2_DB"."sSafetyGate LockRequest" := TRUE;
   END_IF;
   IF #_w3 AND "iSafety door Locking FeedBack_3" THEN
       "ST10_SafetyGate3_DB"."sSafetyGate LockRequest" := TRUE;
   END_IF;
   IF #_w3 AND "iSafety door Locking FeedBack_4" THEN
       "ST10_SafetyGate4_DB"."sSafetyGate LockRequest" := TRUE;
   END_IF;
   IF #_w3 AND "iSafety door Locking FeedBack_5" THEN
       "ST10_SafetyGate5_DB"."sSafetyGate LockRequest" := TRUE;
   END_IF;
   IF #_w3 AND "iSafety door Locking FeedBack_6" THEN
       "ST10_SafetyGate6_DB"."sSafetyGate LockRequest" := TRUE;
   END_IF;
   IF #_w3 AND "iSafety door Locking FeedBack_7" THEN
       "ST10_SafetyGate7_DB"."sSafetyGate LockRequest" := TRUE;
   END_IF;
   IF #_w3 AND "iSafety door Locking FeedBack_8" THEN
       "ST10_SafetyGate8_DB"."sSafetyGate LockRequest" := TRUE;
   END_IF;
   IF #_w3 AND "iSafety Door Locking FeedBack" THEN
       "ST10_SafetyGate9_DB"."sSafetyGate LockRequest" := TRUE;
   END_IF;
   #_w4 := #_w1 AND NOT "Station_Sys".Cmd.Reset;
   #_w5 := #_w4 AND NOT "ST10_GeneralData".P_Plus[48];   // rising edge
   "ST10_GeneralData".P_Plus[48] := #_w4;
   IF #_w5 THEN
       "ST10_SafetyGate1_DB"."sSafetyGate LockRequest" := FALSE;
       "ST10_SafetyGate2_DB"."sSafetyGate LockRequest" := FALSE;
       "ST10_SafetyGate3_DB"."sSafetyGate LockRequest" := FALSE;
       "ST10_SafetyGate4_DB"."sSafetyGate LockRequest" := FALSE;
       "ST10_SafetyGate5_DB"."sSafetyGate LockRequest" := FALSE;
       "ST10_SafetyGate6_DB"."sSafetyGate LockRequest" := FALSE;
       "ST10_SafetyGate7_DB"."sSafetyGate LockRequest" := FALSE;
       "ST10_SafetyGate8_DB"."sSafetyGate LockRequest" := FALSE;
       "ST10_SafetyGate9_DB"."sSafetyGate LockRequest" := FALSE;
   END_IF;
   "ST10_SafetyGate_InterfaceDB".aDev[10].Status."Lock/Unlock Indicator" := "Sys".COM.AlwaysON AND "oSafetyDoorLocked_1" AND "oSafetyDoorLocked_2" AND "oSafetyDoorLocked_3" AND "oSafetyDoorLocked_4" AND "oSafetyDoorLocked_5" AND "oSafetyDoorLocked_6" AND "oSafetyDoorLocked_7" AND "oSafetyDoorLocked_8";
   "ST10_SafetyGate_InterfaceDB".SafetyDoorLamp[10] := "Sys".COM.AlwaysON AND "oSafetyDoorLocked_1" AND "oSafetyDoorLocked_2" AND "oSafetyDoorLocked_3" AND "oSafetyDoorLocked_4" AND "oSafetyDoorLocked_5" AND "oSafetyDoorLocked_6" AND "oSafetyDoorLocked_7" AND "oSafetyDoorLocked_8";
   IF "Sys".COM.AlwaysON AND "oSafetyDoorLocked_1" AND "oSafetyDoorLocked_2" AND "oSafetyDoorLocked_3" AND "oSafetyDoorLocked_4" AND "oSafetyDoorLocked_5" AND "oSafetyDoorLocked_6" AND "oSafetyDoorLocked_7" AND "oSafetyDoorLocked_8" THEN
       "ST10_SafetyGate_InterfaceDB".aDev[10].Status."INT" := 1;
   END_IF;
   IF "Sys".COM.AlwaysON AND NOT "ST10_SafetyGate_InterfaceDB".SafetyDoorLamp[10] THEN
       "ST10_SafetyGate_InterfaceDB".aDev[10].Status."INT" := 3;
   END_IF;
END_REGION

REGION Network 11: E-NG料盒-02安全门锁按钮灯
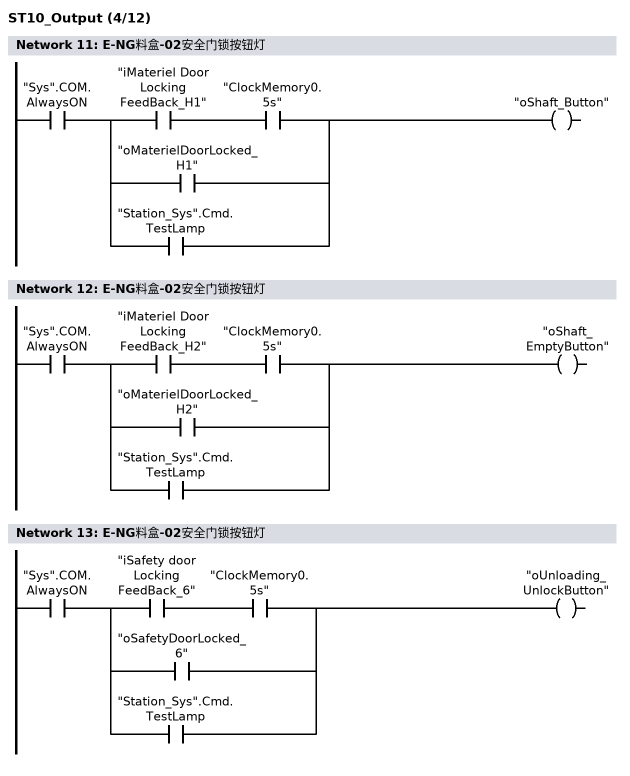
   RUNG wire#powerrail
      Contact( "Sys".COM.AlwaysON )
      wire#w1
      Contact( "iMateriel Door Locking FeedBack_H1" )
      Contact( "ClockMemory0.5s" )
      wire#w2
      Coil( "oShaft_Button" )
   END_RUNG
   RUNG wire#w1
      Contact( "oMaterielDoorLocked_H1" )
   END_RUNG wire#w2
   RUNG wire#w1
      Contact( "Station_Sys".Cmd.TestLamp )
   END_RUNG wire#w2
   // the same network as SCL:
   "oShaft_Button" := "Sys".COM.AlwaysON AND (("iMateriel Door Locking FeedBack_H1" AND "ClockMemory0.5s") OR "oMaterielDoorLocked_H1" OR "Station_Sys".Cmd.TestLamp);
END_REGION

REGION Network 12: E-NG料盒-02安全门锁按钮灯
   RUNG wire#powerrail
      Contact( "Sys".COM.AlwaysON )
      wire#w1
      Contact( "iMateriel Door Locking FeedBack_H2" )
      Contact( "ClockMemory0.5s" )
      wire#w2
      Coil( "oShaft_EmptyButton" )
   END_RUNG
   RUNG wire#w1
      Contact( "oMaterielDoorLocked_H2" )
   END_RUNG wire#w2
   RUNG wire#w1
      Contact( "Station_Sys".Cmd.TestLamp )
   END_RUNG wire#w2
   // the same network as SCL:
   "oShaft_EmptyButton" := "Sys".COM.AlwaysON AND (("iMateriel Door Locking FeedBack_H2" AND "ClockMemory0.5s") OR "oMaterielDoorLocked_H2" OR "Station_Sys".Cmd.TestLamp);
END_REGION

REGION Network 13: E-NG料盒-02安全门锁按钮灯
   RUNG wire#powerrail
      Contact( "Sys".COM.AlwaysON )
      wire#w1
      Contact( "iSafety door Locking FeedBack_6" )
      Contact( "ClockMemory0.5s" )
      wire#w2
      Coil( "oUnloading_UnlockButton" )
   END_RUNG
   RUNG wire#w1
      Contact( "oSafetyDoorLocked_6" )
   END_RUNG wire#w2
   RUNG wire#w1
      Contact( "Station_Sys".Cmd.TestLamp )
   END_RUNG wire#w2
   // the same network as SCL:
   "oUnloading_UnlockButton" := "Sys".COM.AlwaysON AND (("iSafety door Locking FeedBack_6" AND "ClockMemory0.5s") OR "oSafetyDoorLocked_6" OR "Station_Sys".Cmd.TestLamp);
END_REGION

REGION Network 14
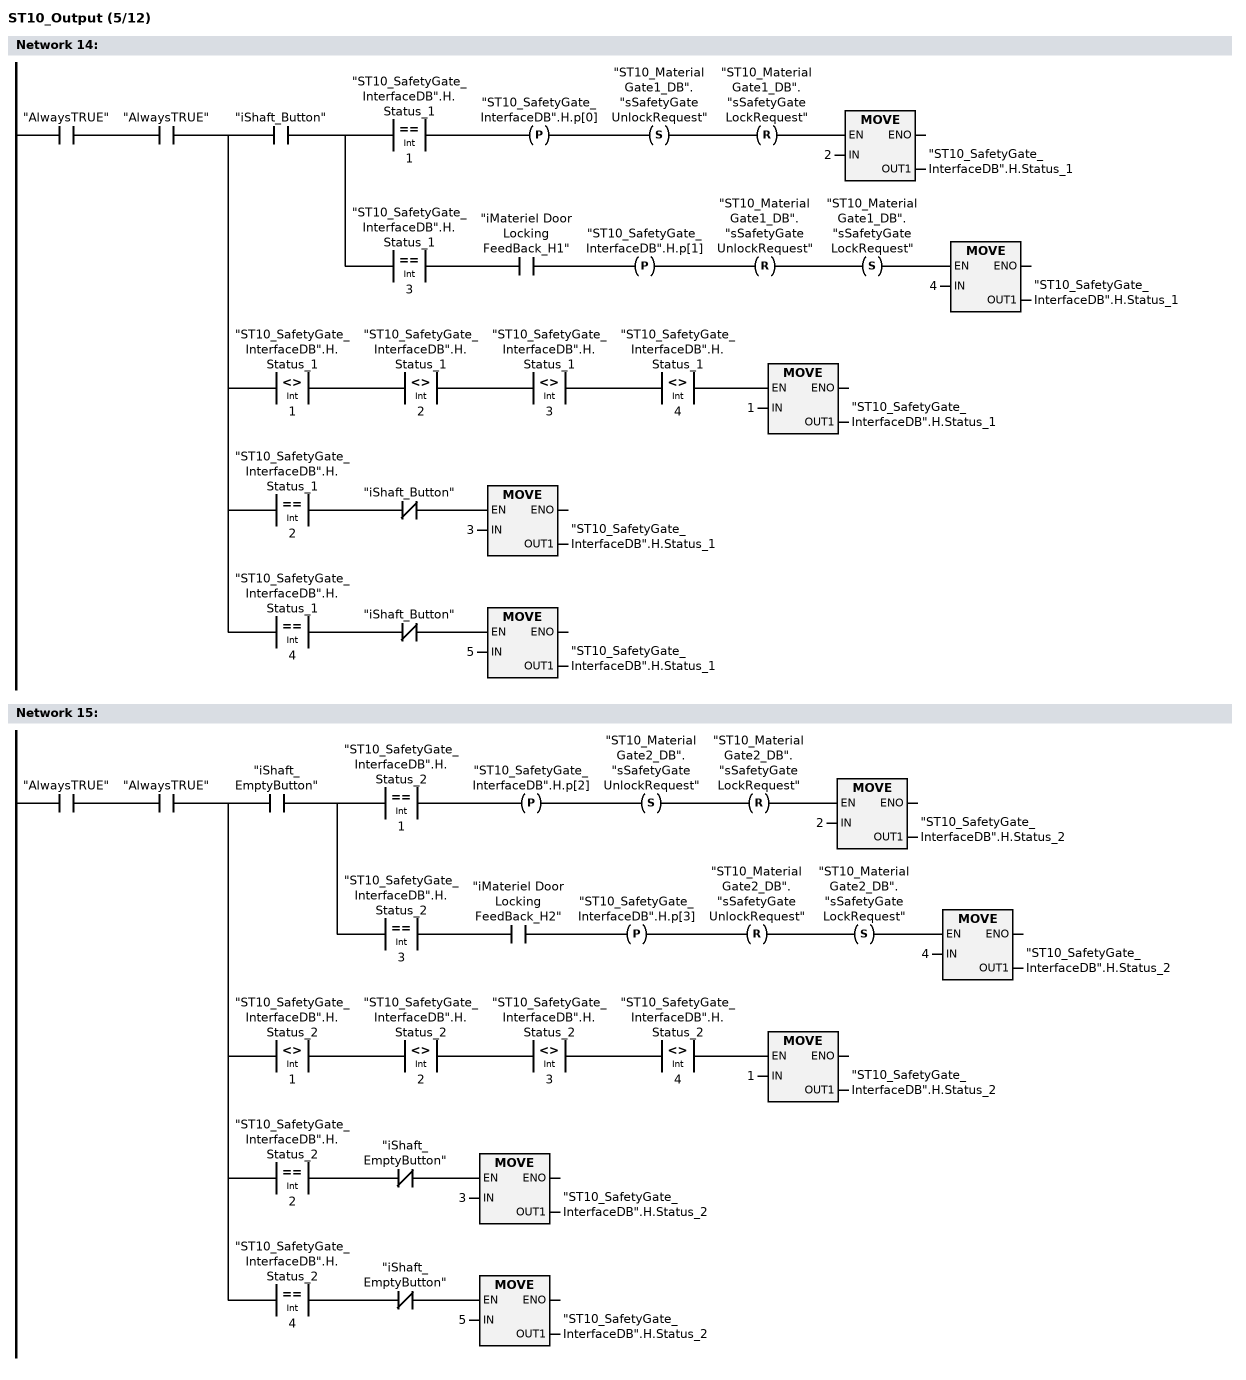
   RUNG wire#powerrail
      Contact( "AlwaysTRUE" )
      Contact( "AlwaysTRUE" )
      wire#w1
      Contact( "iShaft_Button" )
      wire#w2
      { S7_Templates := "SrcType := Int" } EQ_Contact(in1 := "ST10_SafetyGate_InterfaceDB".H.Status_1, in2 := 1)
      P_Trig( "ST10_SafetyGate_InterfaceDB".H.p[0] )
      S_Coil( "ST10_MaterialGate1_DB"."sSafetyGate UnlockRequest" )
      R_Coil( "ST10_MaterialGate1_DB"."sSafetyGate LockRequest" )
      Move(in := 2, out1 => "ST10_SafetyGate_InterfaceDB".H.Status_1)
   END_RUNG
   RUNG wire#w2
      { S7_Templates := "SrcType := Int" } EQ_Contact(in1 := "ST10_SafetyGate_InterfaceDB".H.Status_1, in2 := 3)
      Contact( "iMateriel Door Locking FeedBack_H1" )
      P_Trig( "ST10_SafetyGate_InterfaceDB".H.p[1] )
      R_Coil( "ST10_MaterialGate1_DB"."sSafetyGate UnlockRequest" )
      S_Coil( "ST10_MaterialGate1_DB"."sSafetyGate LockRequest" )
      Move(in := 4, out1 => "ST10_SafetyGate_InterfaceDB".H.Status_1)
   END_RUNG
   RUNG wire#w1
      { S7_Templates := "SrcType := Int" } NE_Contact(in1 := "ST10_SafetyGate_InterfaceDB".H.Status_1, in2 := 1)
      { S7_Templates := "SrcType := Int" } NE_Contact(in1 := "ST10_SafetyGate_InterfaceDB".H.Status_1, in2 := 2)
      { S7_Templates := "SrcType := Int" } NE_Contact(in1 := "ST10_SafetyGate_InterfaceDB".H.Status_1, in2 := 3)
      { S7_Templates := "SrcType := Int" } NE_Contact(in1 := "ST10_SafetyGate_InterfaceDB".H.Status_1, in2 := 4)
      Move(in := 1, out1 => "ST10_SafetyGate_InterfaceDB".H.Status_1)
   END_RUNG
   RUNG wire#w1
      { S7_Templates := "SrcType := Int" } EQ_Contact(in1 := "ST10_SafetyGate_InterfaceDB".H.Status_1, in2 := 2)
      I_Contact( "iShaft_Button" )
      Move(in := 3, out1 => "ST10_SafetyGate_InterfaceDB".H.Status_1)
   END_RUNG
   RUNG wire#w1
      { S7_Templates := "SrcType := Int" } EQ_Contact(in1 := "ST10_SafetyGate_InterfaceDB".H.Status_1, in2 := 4)
      I_Contact( "iShaft_Button" )
      Move(in := 5, out1 => "ST10_SafetyGate_InterfaceDB".H.Status_1)
   END_RUNG
   // the same network as SCL:
   #_w1 := "AlwaysTRUE" AND "AlwaysTRUE";
   #_w2 := #_w1 AND "iShaft_Button";
   #_w3 := #_w2 AND ("ST10_SafetyGate_InterfaceDB".H.Status_1 = 1);
   #_w4 := #_w3 AND NOT "ST10_SafetyGate_InterfaceDB".H.p[0];   // rising edge
   "ST10_SafetyGate_InterfaceDB".H.p[0] := #_w3;
   IF #_w4 THEN
       "ST10_MaterialGate1_DB"."sSafetyGate UnlockRequest" := TRUE;
       "ST10_MaterialGate1_DB"."sSafetyGate LockRequest" := FALSE;
       "ST10_SafetyGate_InterfaceDB".H.Status_1 := 2;
   END_IF;
   #_w5 := #_w2 AND ("ST10_SafetyGate_InterfaceDB".H.Status_1 = 3) AND "iMateriel Door Locking FeedBack_H1";
   #_w6 := #_w5 AND NOT "ST10_SafetyGate_InterfaceDB".H.p[1];   // rising edge
   "ST10_SafetyGate_InterfaceDB".H.p[1] := #_w5;
   IF #_w6 THEN
       "ST10_MaterialGate1_DB"."sSafetyGate UnlockRequest" := FALSE;
       "ST10_MaterialGate1_DB"."sSafetyGate LockRequest" := TRUE;
       "ST10_SafetyGate_InterfaceDB".H.Status_1 := 4;
   END_IF;
   IF #_w1 AND ("ST10_SafetyGate_InterfaceDB".H.Status_1 <> 1) AND ("ST10_SafetyGate_InterfaceDB".H.Status_1 <> 2) AND ("ST10_SafetyGate_InterfaceDB".H.Status_1 <> 3) AND ("ST10_SafetyGate_InterfaceDB".H.Status_1 <> 4) THEN
       "ST10_SafetyGate_InterfaceDB".H.Status_1 := 1;
   END_IF;
   IF #_w1 AND ("ST10_SafetyGate_InterfaceDB".H.Status_1 = 2) AND NOT "iShaft_Button" THEN
       "ST10_SafetyGate_InterfaceDB".H.Status_1 := 3;
   END_IF;
   IF #_w1 AND ("ST10_SafetyGate_InterfaceDB".H.Status_1 = 4) AND NOT "iShaft_Button" THEN
       "ST10_SafetyGate_InterfaceDB".H.Status_1 := 5;
   END_IF;
END_REGION

REGION Network 15
   RUNG wire#powerrail
      Contact( "AlwaysTRUE" )
      Contact( "AlwaysTRUE" )
      wire#w1
      Contact( "iShaft_EmptyButton" )
      wire#w2
      { S7_Templates := "SrcType := Int" } EQ_Contact(in1 := "ST10_SafetyGate_InterfaceDB".H.Status_2, in2 := 1)
      P_Trig( "ST10_SafetyGate_InterfaceDB".H.p[2] )
      S_Coil( "ST10_MaterialGate2_DB"."sSafetyGate UnlockRequest" )
      R_Coil( "ST10_MaterialGate2_DB"."sSafetyGate LockRequest" )
      Move(in := 2, out1 => "ST10_SafetyGate_InterfaceDB".H.Status_2)
   END_RUNG
   RUNG wire#w2
      { S7_Templates := "SrcType := Int" } EQ_Contact(in1 := "ST10_SafetyGate_InterfaceDB".H.Status_2, in2 := 3)
      Contact( "iMateriel Door Locking FeedBack_H2" )
      P_Trig( "ST10_SafetyGate_InterfaceDB".H.p[3] )
      R_Coil( "ST10_MaterialGate2_DB"."sSafetyGate UnlockRequest" )
      S_Coil( "ST10_MaterialGate2_DB"."sSafetyGate LockRequest" )
      Move(in := 4, out1 => "ST10_SafetyGate_InterfaceDB".H.Status_2)
   END_RUNG
   RUNG wire#w1
      { S7_Templates := "SrcType := Int" } NE_Contact(in1 := "ST10_SafetyGate_InterfaceDB".H.Status_2, in2 := 1)
      { S7_Templates := "SrcType := Int" } NE_Contact(in1 := "ST10_SafetyGate_InterfaceDB".H.Status_2, in2 := 2)
      { S7_Templates := "SrcType := Int" } NE_Contact(in1 := "ST10_SafetyGate_InterfaceDB".H.Status_2, in2 := 3)
      { S7_Templates := "SrcType := Int" } NE_Contact(in1 := "ST10_SafetyGate_InterfaceDB".H.Status_2, in2 := 4)
      Move(in := 1, out1 => "ST10_SafetyGate_InterfaceDB".H.Status_2)
   END_RUNG
   RUNG wire#w1
      { S7_Templates := "SrcType := Int" } EQ_Contact(in1 := "ST10_SafetyGate_InterfaceDB".H.Status_2, in2 := 2)
      I_Contact( "iShaft_EmptyButton" )
      Move(in := 3, out1 => "ST10_SafetyGate_InterfaceDB".H.Status_2)
   END_RUNG
   RUNG wire#w1
      { S7_Templates := "SrcType := Int" } EQ_Contact(in1 := "ST10_SafetyGate_InterfaceDB".H.Status_2, in2 := 4)
      I_Contact( "iShaft_EmptyButton" )
      Move(in := 5, out1 => "ST10_SafetyGate_InterfaceDB".H.Status_2)
   END_RUNG
   // the same network as SCL:
   #_w1 := "AlwaysTRUE" AND "AlwaysTRUE";
   #_w2 := #_w1 AND "iShaft_EmptyButton";
   #_w3 := #_w2 AND ("ST10_SafetyGate_InterfaceDB".H.Status_2 = 1);
   #_w4 := #_w3 AND NOT "ST10_SafetyGate_InterfaceDB".H.p[2];   // rising edge
   "ST10_SafetyGate_InterfaceDB".H.p[2] := #_w3;
   IF #_w4 THEN
       "ST10_MaterialGate2_DB"."sSafetyGate UnlockRequest" := TRUE;
       "ST10_MaterialGate2_DB"."sSafetyGate LockRequest" := FALSE;
       "ST10_SafetyGate_InterfaceDB".H.Status_2 := 2;
   END_IF;
   #_w5 := #_w2 AND ("ST10_SafetyGate_InterfaceDB".H.Status_2 = 3) AND "iMateriel Door Locking FeedBack_H2";
   #_w6 := #_w5 AND NOT "ST10_SafetyGate_InterfaceDB".H.p[3];   // rising edge
   "ST10_SafetyGate_InterfaceDB".H.p[3] := #_w5;
   IF #_w6 THEN
       "ST10_MaterialGate2_DB"."sSafetyGate UnlockRequest" := FALSE;
       "ST10_MaterialGate2_DB"."sSafetyGate LockRequest" := TRUE;
       "ST10_SafetyGate_InterfaceDB".H.Status_2 := 4;
   END_IF;
   IF #_w1 AND ("ST10_SafetyGate_InterfaceDB".H.Status_2 <> 1) AND ("ST10_SafetyGate_InterfaceDB".H.Status_2 <> 2) AND ("ST10_SafetyGate_InterfaceDB".H.Status_2 <> 3) AND ("ST10_SafetyGate_InterfaceDB".H.Status_2 <> 4) THEN
       "ST10_SafetyGate_InterfaceDB".H.Status_2 := 1;
   END_IF;
   IF #_w1 AND ("ST10_SafetyGate_InterfaceDB".H.Status_2 = 2) AND NOT "iShaft_EmptyButton" THEN
       "ST10_SafetyGate_InterfaceDB".H.Status_2 := 3;
   END_IF;
   IF #_w1 AND ("ST10_SafetyGate_InterfaceDB".H.Status_2 = 4) AND NOT "iShaft_EmptyButton" THEN
       "ST10_SafetyGate_InterfaceDB".H.Status_2 := 5;
   END_IF;
END_REGION

REGION Network 16
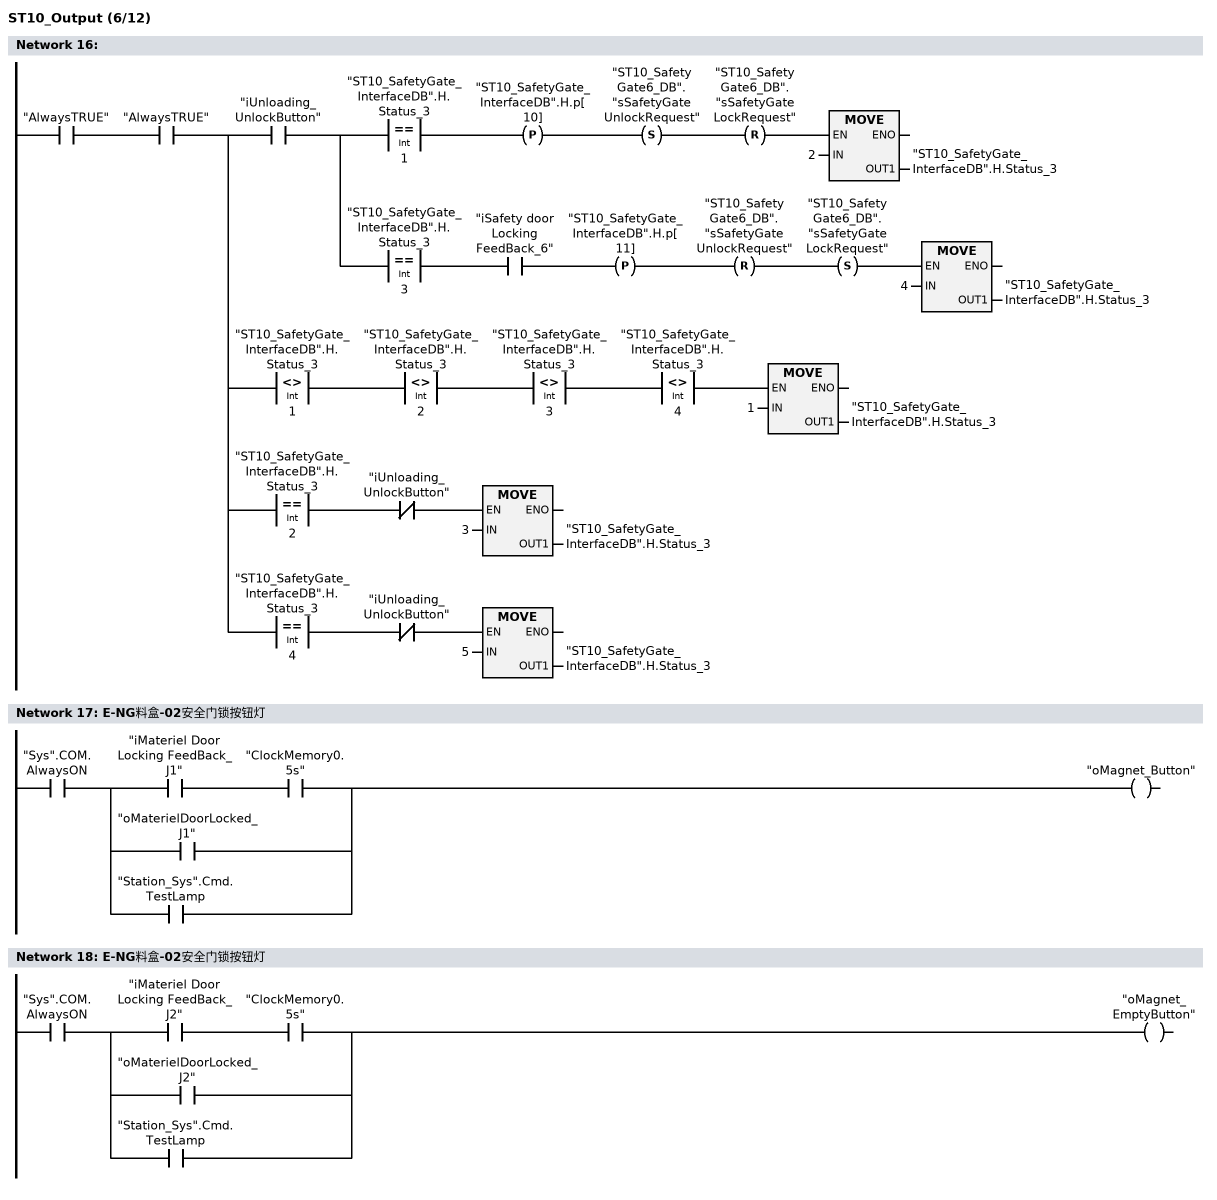
   RUNG wire#powerrail
      Contact( "AlwaysTRUE" )
      Contact( "AlwaysTRUE" )
      wire#w1
      Contact( "iUnloading_UnlockButton" )
      wire#w2
      { S7_Templates := "SrcType := Int" } EQ_Contact(in1 := "ST10_SafetyGate_InterfaceDB".H.Status_3, in2 := 1)
      P_Trig( "ST10_SafetyGate_InterfaceDB".H.p[10] )
      S_Coil( "ST10_SafetyGate6_DB"."sSafetyGate UnlockRequest" )
      R_Coil( "ST10_SafetyGate6_DB"."sSafetyGate LockRequest" )
      Move(in := 2, out1 => "ST10_SafetyGate_InterfaceDB".H.Status_3)
   END_RUNG
   RUNG wire#w2
      { S7_Templates := "SrcType := Int" } EQ_Contact(in1 := "ST10_SafetyGate_InterfaceDB".H.Status_3, in2 := 3)
      Contact( "iSafety door Locking FeedBack_6" )
      P_Trig( "ST10_SafetyGate_InterfaceDB".H.p[11] )
      R_Coil( "ST10_SafetyGate6_DB"."sSafetyGate UnlockRequest" )
      S_Coil( "ST10_SafetyGate6_DB"."sSafetyGate LockRequest" )
      Move(in := 4, out1 => "ST10_SafetyGate_InterfaceDB".H.Status_3)
   END_RUNG
   RUNG wire#w1
      { S7_Templates := "SrcType := Int" } NE_Contact(in1 := "ST10_SafetyGate_InterfaceDB".H.Status_3, in2 := 1)
      { S7_Templates := "SrcType := Int" } NE_Contact(in1 := "ST10_SafetyGate_InterfaceDB".H.Status_3, in2 := 2)
      { S7_Templates := "SrcType := Int" } NE_Contact(in1 := "ST10_SafetyGate_InterfaceDB".H.Status_3, in2 := 3)
      { S7_Templates := "SrcType := Int" } NE_Contact(in1 := "ST10_SafetyGate_InterfaceDB".H.Status_3, in2 := 4)
      Move(in := 1, out1 => "ST10_SafetyGate_InterfaceDB".H.Status_3)
   END_RUNG
   RUNG wire#w1
      { S7_Templates := "SrcType := Int" } EQ_Contact(in1 := "ST10_SafetyGate_InterfaceDB".H.Status_3, in2 := 2)
      I_Contact( "iUnloading_UnlockButton" )
      Move(in := 3, out1 => "ST10_SafetyGate_InterfaceDB".H.Status_3)
   END_RUNG
   RUNG wire#w1
      { S7_Templates := "SrcType := Int" } EQ_Contact(in1 := "ST10_SafetyGate_InterfaceDB".H.Status_3, in2 := 4)
      I_Contact( "iUnloading_UnlockButton" )
      Move(in := 5, out1 => "ST10_SafetyGate_InterfaceDB".H.Status_3)
   END_RUNG
   // the same network as SCL:
   #_w1 := "AlwaysTRUE" AND "AlwaysTRUE";
   #_w2 := #_w1 AND "iUnloading_UnlockButton";
   #_w3 := #_w2 AND ("ST10_SafetyGate_InterfaceDB".H.Status_3 = 1);
   #_w4 := #_w3 AND NOT "ST10_SafetyGate_InterfaceDB".H.p[10];   // rising edge
   "ST10_SafetyGate_InterfaceDB".H.p[10] := #_w3;
   IF #_w4 THEN
       "ST10_SafetyGate6_DB"."sSafetyGate UnlockRequest" := TRUE;
       "ST10_SafetyGate6_DB"."sSafetyGate LockRequest" := FALSE;
       "ST10_SafetyGate_InterfaceDB".H.Status_3 := 2;
   END_IF;
   #_w5 := #_w2 AND ("ST10_SafetyGate_InterfaceDB".H.Status_3 = 3) AND "iSafety door Locking FeedBack_6";
   #_w6 := #_w5 AND NOT "ST10_SafetyGate_InterfaceDB".H.p[11];   // rising edge
   "ST10_SafetyGate_InterfaceDB".H.p[11] := #_w5;
   IF #_w6 THEN
       "ST10_SafetyGate6_DB"."sSafetyGate UnlockRequest" := FALSE;
       "ST10_SafetyGate6_DB"."sSafetyGate LockRequest" := TRUE;
       "ST10_SafetyGate_InterfaceDB".H.Status_3 := 4;
   END_IF;
   IF #_w1 AND ("ST10_SafetyGate_InterfaceDB".H.Status_3 <> 1) AND ("ST10_SafetyGate_InterfaceDB".H.Status_3 <> 2) AND ("ST10_SafetyGate_InterfaceDB".H.Status_3 <> 3) AND ("ST10_SafetyGate_InterfaceDB".H.Status_3 <> 4) THEN
       "ST10_SafetyGate_InterfaceDB".H.Status_3 := 1;
   END_IF;
   IF #_w1 AND ("ST10_SafetyGate_InterfaceDB".H.Status_3 = 2) AND NOT "iUnloading_UnlockButton" THEN
       "ST10_SafetyGate_InterfaceDB".H.Status_3 := 3;
   END_IF;
   IF #_w1 AND ("ST10_SafetyGate_InterfaceDB".H.Status_3 = 4) AND NOT "iUnloading_UnlockButton" THEN
       "ST10_SafetyGate_InterfaceDB".H.Status_3 := 5;
   END_IF;
END_REGION

REGION Network 17: E-NG料盒-02安全门锁按钮灯
   RUNG wire#powerrail
      Contact( "Sys".COM.AlwaysON )
      wire#w1
      Contact( "iMateriel Door Locking FeedBack_J1" )
      Contact( "ClockMemory0.5s" )
      wire#w2
      Coil( "oMagnet_Button" )
   END_RUNG
   RUNG wire#w1
      Contact( "oMaterielDoorLocked_J1" )
   END_RUNG wire#w2
   RUNG wire#w1
      Contact( "Station_Sys".Cmd.TestLamp )
   END_RUNG wire#w2
   // the same network as SCL:
   "oMagnet_Button" := "Sys".COM.AlwaysON AND (("iMateriel Door Locking FeedBack_J1" AND "ClockMemory0.5s") OR "oMaterielDoorLocked_J1" OR "Station_Sys".Cmd.TestLamp);
END_REGION

REGION Network 18: E-NG料盒-02安全门锁按钮灯
   RUNG wire#powerrail
      Contact( "Sys".COM.AlwaysON )
      wire#w1
      Contact( "iMateriel Door Locking FeedBack_J2" )
      Contact( "ClockMemory0.5s" )
      wire#w2
      Coil( "oMagnet_EmptyButton" )
   END_RUNG
   RUNG wire#w1
      Contact( "oMaterielDoorLocked_J2" )
   END_RUNG wire#w2
   RUNG wire#w1
      Contact( "Station_Sys".Cmd.TestLamp )
   END_RUNG wire#w2
   // the same network as SCL:
   "oMagnet_EmptyButton" := "Sys".COM.AlwaysON AND (("iMateriel Door Locking FeedBack_J2" AND "ClockMemory0.5s") OR "oMaterielDoorLocked_J2" OR "Station_Sys".Cmd.TestLamp);
END_REGION

REGION Network 19: E-NG料盒-02安全门锁按钮灯
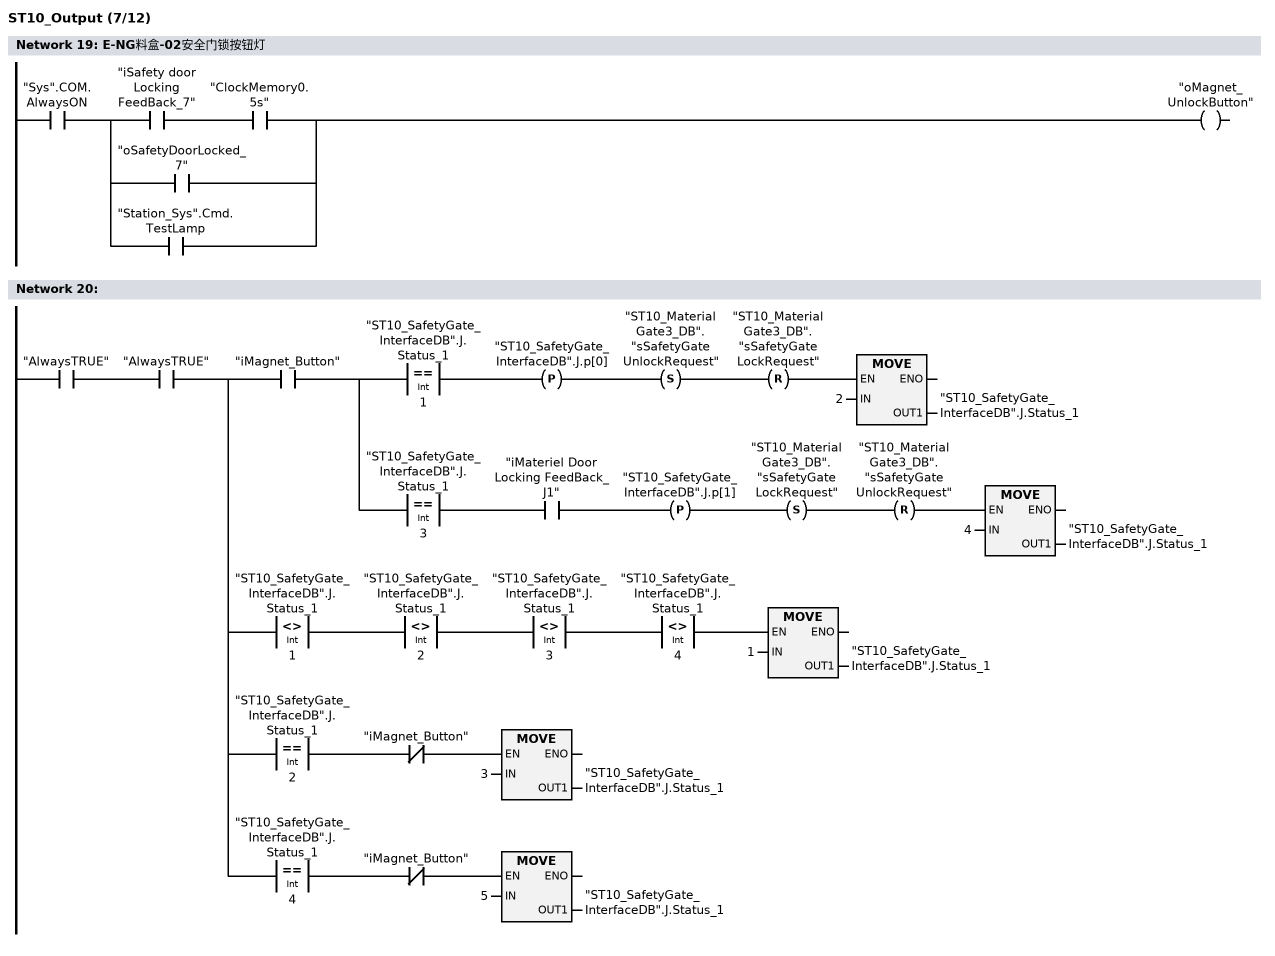
   RUNG wire#powerrail
      Contact( "Sys".COM.AlwaysON )
      wire#w1
      Contact( "iSafety door Locking FeedBack_7" )
      Contact( "ClockMemory0.5s" )
      wire#w2
      Coil( "oMagnet_UnlockButton" )
   END_RUNG
   RUNG wire#w1
      Contact( "oSafetyDoorLocked_7" )
   END_RUNG wire#w2
   RUNG wire#w1
      Contact( "Station_Sys".Cmd.TestLamp )
   END_RUNG wire#w2
   // the same network as SCL:
   "oMagnet_UnlockButton" := "Sys".COM.AlwaysON AND (("iSafety door Locking FeedBack_7" AND "ClockMemory0.5s") OR "oSafetyDoorLocked_7" OR "Station_Sys".Cmd.TestLamp);
END_REGION

REGION Network 20
   RUNG wire#powerrail
      Contact( "AlwaysTRUE" )
      Contact( "AlwaysTRUE" )
      wire#w1
      Contact( "iMagnet_Button" )
      wire#w2
      { S7_Templates := "SrcType := Int" } EQ_Contact(in1 := "ST10_SafetyGate_InterfaceDB".J.Status_1, in2 := 1)
      P_Trig( "ST10_SafetyGate_InterfaceDB".J.p[0] )
      S_Coil( "ST10_MaterialGate3_DB"."sSafetyGate UnlockRequest" )
      R_Coil( "ST10_MaterialGate3_DB"."sSafetyGate LockRequest" )
      Move(in := 2, out1 => "ST10_SafetyGate_InterfaceDB".J.Status_1)
   END_RUNG
   RUNG wire#w2
      { S7_Templates := "SrcType := Int" } EQ_Contact(in1 := "ST10_SafetyGate_InterfaceDB".J.Status_1, in2 := 3)
      Contact( "iMateriel Door Locking FeedBack_J1" )
      P_Trig( "ST10_SafetyGate_InterfaceDB".J.p[1] )
      S_Coil( "ST10_MaterialGate3_DB"."sSafetyGate LockRequest" )
      R_Coil( "ST10_MaterialGate3_DB"."sSafetyGate UnlockRequest" )
      Move(in := 4, out1 => "ST10_SafetyGate_InterfaceDB".J.Status_1)
   END_RUNG
   RUNG wire#w1
      { S7_Templates := "SrcType := Int" } NE_Contact(in1 := "ST10_SafetyGate_InterfaceDB".J.Status_1, in2 := 1)
      { S7_Templates := "SrcType := Int" } NE_Contact(in1 := "ST10_SafetyGate_InterfaceDB".J.Status_1, in2 := 2)
      { S7_Templates := "SrcType := Int" } NE_Contact(in1 := "ST10_SafetyGate_InterfaceDB".J.Status_1, in2 := 3)
      { S7_Templates := "SrcType := Int" } NE_Contact(in1 := "ST10_SafetyGate_InterfaceDB".J.Status_1, in2 := 4)
      Move(in := 1, out1 => "ST10_SafetyGate_InterfaceDB".J.Status_1)
   END_RUNG
   RUNG wire#w1
      { S7_Templates := "SrcType := Int" } EQ_Contact(in1 := "ST10_SafetyGate_InterfaceDB".J.Status_1, in2 := 2)
      I_Contact( "iMagnet_Button" )
      Move(in := 3, out1 => "ST10_SafetyGate_InterfaceDB".J.Status_1)
   END_RUNG
   RUNG wire#w1
      { S7_Templates := "SrcType := Int" } EQ_Contact(in1 := "ST10_SafetyGate_InterfaceDB".J.Status_1, in2 := 4)
      I_Contact( "iMagnet_Button" )
      Move(in := 5, out1 => "ST10_SafetyGate_InterfaceDB".J.Status_1)
   END_RUNG
   // the same network as SCL:
   #_w1 := "AlwaysTRUE" AND "AlwaysTRUE";
   #_w2 := #_w1 AND "iMagnet_Button";
   #_w3 := #_w2 AND ("ST10_SafetyGate_InterfaceDB".J.Status_1 = 1);
   #_w4 := #_w3 AND NOT "ST10_SafetyGate_InterfaceDB".J.p[0];   // rising edge
   "ST10_SafetyGate_InterfaceDB".J.p[0] := #_w3;
   IF #_w4 THEN
       "ST10_MaterialGate3_DB"."sSafetyGate UnlockRequest" := TRUE;
       "ST10_MaterialGate3_DB"."sSafetyGate LockRequest" := FALSE;
       "ST10_SafetyGate_InterfaceDB".J.Status_1 := 2;
   END_IF;
   #_w5 := #_w2 AND ("ST10_SafetyGate_InterfaceDB".J.Status_1 = 3) AND "iMateriel Door Locking FeedBack_J1";
   #_w6 := #_w5 AND NOT "ST10_SafetyGate_InterfaceDB".J.p[1];   // rising edge
   "ST10_SafetyGate_InterfaceDB".J.p[1] := #_w5;
   IF #_w6 THEN
       "ST10_MaterialGate3_DB"."sSafetyGate LockRequest" := TRUE;
       "ST10_MaterialGate3_DB"."sSafetyGate UnlockRequest" := FALSE;
       "ST10_SafetyGate_InterfaceDB".J.Status_1 := 4;
   END_IF;
   IF #_w1 AND ("ST10_SafetyGate_InterfaceDB".J.Status_1 <> 1) AND ("ST10_SafetyGate_InterfaceDB".J.Status_1 <> 2) AND ("ST10_SafetyGate_InterfaceDB".J.Status_1 <> 3) AND ("ST10_SafetyGate_InterfaceDB".J.Status_1 <> 4) THEN
       "ST10_SafetyGate_InterfaceDB".J.Status_1 := 1;
   END_IF;
   IF #_w1 AND ("ST10_SafetyGate_InterfaceDB".J.Status_1 = 2) AND NOT "iMagnet_Button" THEN
       "ST10_SafetyGate_InterfaceDB".J.Status_1 := 3;
   END_IF;
   IF #_w1 AND ("ST10_SafetyGate_InterfaceDB".J.Status_1 = 4) AND NOT "iMagnet_Button" THEN
       "ST10_SafetyGate_InterfaceDB".J.Status_1 := 5;
   END_IF;
END_REGION

REGION Network 21
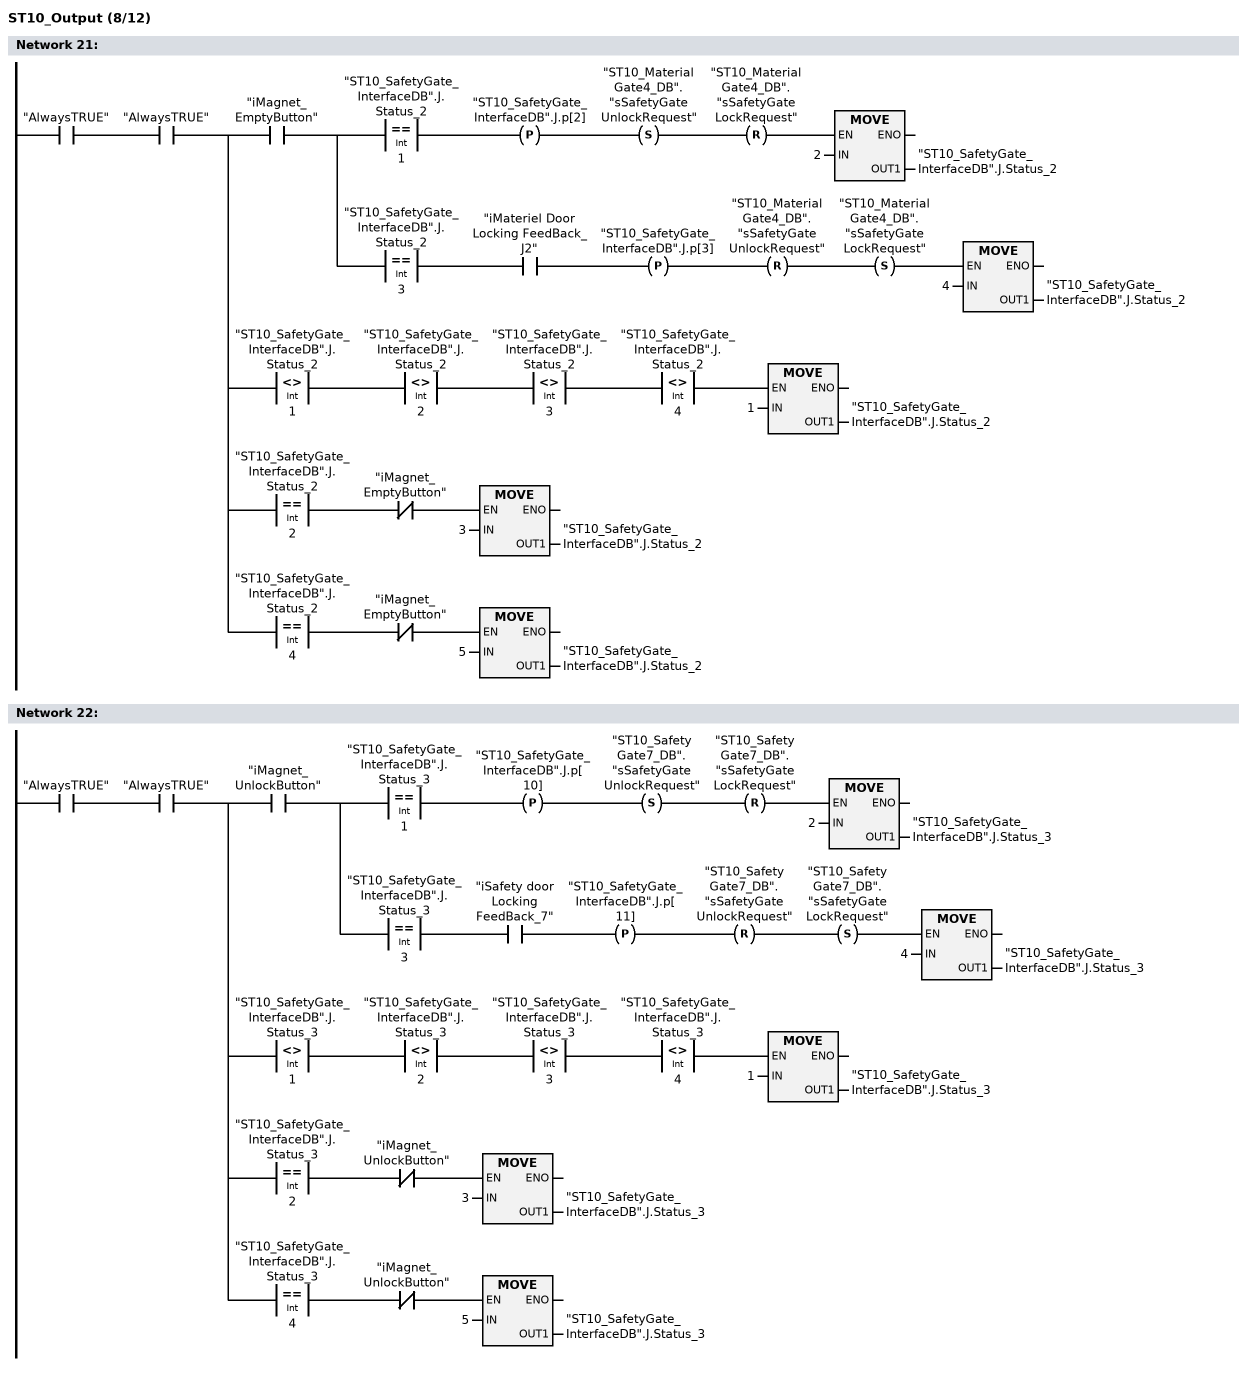
   RUNG wire#powerrail
      Contact( "AlwaysTRUE" )
      Contact( "AlwaysTRUE" )
      wire#w1
      Contact( "iMagnet_EmptyButton" )
      wire#w2
      { S7_Templates := "SrcType := Int" } EQ_Contact(in1 := "ST10_SafetyGate_InterfaceDB".J.Status_2, in2 := 1)
      P_Trig( "ST10_SafetyGate_InterfaceDB".J.p[2] )
      S_Coil( "ST10_MaterialGate4_DB"."sSafetyGate UnlockRequest" )
      R_Coil( "ST10_MaterialGate4_DB"."sSafetyGate LockRequest" )
      Move(in := 2, out1 => "ST10_SafetyGate_InterfaceDB".J.Status_2)
   END_RUNG
   RUNG wire#w2
      { S7_Templates := "SrcType := Int" } EQ_Contact(in1 := "ST10_SafetyGate_InterfaceDB".J.Status_2, in2 := 3)
      Contact( "iMateriel Door Locking FeedBack_J2" )
      P_Trig( "ST10_SafetyGate_InterfaceDB".J.p[3] )
      R_Coil( "ST10_MaterialGate4_DB"."sSafetyGate UnlockRequest" )
      S_Coil( "ST10_MaterialGate4_DB"."sSafetyGate LockRequest" )
      Move(in := 4, out1 => "ST10_SafetyGate_InterfaceDB".J.Status_2)
   END_RUNG
   RUNG wire#w1
      { S7_Templates := "SrcType := Int" } NE_Contact(in1 := "ST10_SafetyGate_InterfaceDB".J.Status_2, in2 := 1)
      { S7_Templates := "SrcType := Int" } NE_Contact(in1 := "ST10_SafetyGate_InterfaceDB".J.Status_2, in2 := 2)
      { S7_Templates := "SrcType := Int" } NE_Contact(in1 := "ST10_SafetyGate_InterfaceDB".J.Status_2, in2 := 3)
      { S7_Templates := "SrcType := Int" } NE_Contact(in1 := "ST10_SafetyGate_InterfaceDB".J.Status_2, in2 := 4)
      Move(in := 1, out1 => "ST10_SafetyGate_InterfaceDB".J.Status_2)
   END_RUNG
   RUNG wire#w1
      { S7_Templates := "SrcType := Int" } EQ_Contact(in1 := "ST10_SafetyGate_InterfaceDB".J.Status_2, in2 := 2)
      I_Contact( "iMagnet_EmptyButton" )
      Move(in := 3, out1 => "ST10_SafetyGate_InterfaceDB".J.Status_2)
   END_RUNG
   RUNG wire#w1
      { S7_Templates := "SrcType := Int" } EQ_Contact(in1 := "ST10_SafetyGate_InterfaceDB".J.Status_2, in2 := 4)
      I_Contact( "iMagnet_EmptyButton" )
      Move(in := 5, out1 => "ST10_SafetyGate_InterfaceDB".J.Status_2)
   END_RUNG
   // the same network as SCL:
   #_w1 := "AlwaysTRUE" AND "AlwaysTRUE";
   #_w2 := #_w1 AND "iMagnet_EmptyButton";
   #_w3 := #_w2 AND ("ST10_SafetyGate_InterfaceDB".J.Status_2 = 1);
   #_w4 := #_w3 AND NOT "ST10_SafetyGate_InterfaceDB".J.p[2];   // rising edge
   "ST10_SafetyGate_InterfaceDB".J.p[2] := #_w3;
   IF #_w4 THEN
       "ST10_MaterialGate4_DB"."sSafetyGate UnlockRequest" := TRUE;
       "ST10_MaterialGate4_DB"."sSafetyGate LockRequest" := FALSE;
       "ST10_SafetyGate_InterfaceDB".J.Status_2 := 2;
   END_IF;
   #_w5 := #_w2 AND ("ST10_SafetyGate_InterfaceDB".J.Status_2 = 3) AND "iMateriel Door Locking FeedBack_J2";
   #_w6 := #_w5 AND NOT "ST10_SafetyGate_InterfaceDB".J.p[3];   // rising edge
   "ST10_SafetyGate_InterfaceDB".J.p[3] := #_w5;
   IF #_w6 THEN
       "ST10_MaterialGate4_DB"."sSafetyGate UnlockRequest" := FALSE;
       "ST10_MaterialGate4_DB"."sSafetyGate LockRequest" := TRUE;
       "ST10_SafetyGate_InterfaceDB".J.Status_2 := 4;
   END_IF;
   IF #_w1 AND ("ST10_SafetyGate_InterfaceDB".J.Status_2 <> 1) AND ("ST10_SafetyGate_InterfaceDB".J.Status_2 <> 2) AND ("ST10_SafetyGate_InterfaceDB".J.Status_2 <> 3) AND ("ST10_SafetyGate_InterfaceDB".J.Status_2 <> 4) THEN
       "ST10_SafetyGate_InterfaceDB".J.Status_2 := 1;
   END_IF;
   IF #_w1 AND ("ST10_SafetyGate_InterfaceDB".J.Status_2 = 2) AND NOT "iMagnet_EmptyButton" THEN
       "ST10_SafetyGate_InterfaceDB".J.Status_2 := 3;
   END_IF;
   IF #_w1 AND ("ST10_SafetyGate_InterfaceDB".J.Status_2 = 4) AND NOT "iMagnet_EmptyButton" THEN
       "ST10_SafetyGate_InterfaceDB".J.Status_2 := 5;
   END_IF;
END_REGION

REGION Network 22
   RUNG wire#powerrail
      Contact( "AlwaysTRUE" )
      Contact( "AlwaysTRUE" )
      wire#w1
      Contact( "iMagnet_UnlockButton" )
      wire#w2
      { S7_Templates := "SrcType := Int" } EQ_Contact(in1 := "ST10_SafetyGate_InterfaceDB".J.Status_3, in2 := 1)
      P_Trig( "ST10_SafetyGate_InterfaceDB".J.p[10] )
      S_Coil( "ST10_SafetyGate7_DB"."sSafetyGate UnlockRequest" )
      R_Coil( "ST10_SafetyGate7_DB"."sSafetyGate LockRequest" )
      Move(in := 2, out1 => "ST10_SafetyGate_InterfaceDB".J.Status_3)
   END_RUNG
   RUNG wire#w2
      { S7_Templates := "SrcType := Int" } EQ_Contact(in1 := "ST10_SafetyGate_InterfaceDB".J.Status_3, in2 := 3)
      Contact( "iSafety door Locking FeedBack_7" )
      P_Trig( "ST10_SafetyGate_InterfaceDB".J.p[11] )
      R_Coil( "ST10_SafetyGate7_DB"."sSafetyGate UnlockRequest" )
      S_Coil( "ST10_SafetyGate7_DB"."sSafetyGate LockRequest" )
      Move(in := 4, out1 => "ST10_SafetyGate_InterfaceDB".J.Status_3)
   END_RUNG
   RUNG wire#w1
      { S7_Templates := "SrcType := Int" } NE_Contact(in1 := "ST10_SafetyGate_InterfaceDB".J.Status_3, in2 := 1)
      { S7_Templates := "SrcType := Int" } NE_Contact(in1 := "ST10_SafetyGate_InterfaceDB".J.Status_3, in2 := 2)
      { S7_Templates := "SrcType := Int" } NE_Contact(in1 := "ST10_SafetyGate_InterfaceDB".J.Status_3, in2 := 3)
      { S7_Templates := "SrcType := Int" } NE_Contact(in1 := "ST10_SafetyGate_InterfaceDB".J.Status_3, in2 := 4)
      Move(in := 1, out1 => "ST10_SafetyGate_InterfaceDB".J.Status_3)
   END_RUNG
   RUNG wire#w1
      { S7_Templates := "SrcType := Int" } EQ_Contact(in1 := "ST10_SafetyGate_InterfaceDB".J.Status_3, in2 := 2)
      I_Contact( "iMagnet_UnlockButton" )
      Move(in := 3, out1 => "ST10_SafetyGate_InterfaceDB".J.Status_3)
   END_RUNG
   RUNG wire#w1
      { S7_Templates := "SrcType := Int" } EQ_Contact(in1 := "ST10_SafetyGate_InterfaceDB".J.Status_3, in2 := 4)
      I_Contact( "iMagnet_UnlockButton" )
      Move(in := 5, out1 => "ST10_SafetyGate_InterfaceDB".J.Status_3)
   END_RUNG
   // the same network as SCL:
   #_w1 := "AlwaysTRUE" AND "AlwaysTRUE";
   #_w2 := #_w1 AND "iMagnet_UnlockButton";
   #_w3 := #_w2 AND ("ST10_SafetyGate_InterfaceDB".J.Status_3 = 1);
   #_w4 := #_w3 AND NOT "ST10_SafetyGate_InterfaceDB".J.p[10];   // rising edge
   "ST10_SafetyGate_InterfaceDB".J.p[10] := #_w3;
   IF #_w4 THEN
       "ST10_SafetyGate7_DB"."sSafetyGate UnlockRequest" := TRUE;
       "ST10_SafetyGate7_DB"."sSafetyGate LockRequest" := FALSE;
       "ST10_SafetyGate_InterfaceDB".J.Status_3 := 2;
   END_IF;
   #_w5 := #_w2 AND ("ST10_SafetyGate_InterfaceDB".J.Status_3 = 3) AND "iSafety door Locking FeedBack_7";
   #_w6 := #_w5 AND NOT "ST10_SafetyGate_InterfaceDB".J.p[11];   // rising edge
   "ST10_SafetyGate_InterfaceDB".J.p[11] := #_w5;
   IF #_w6 THEN
       "ST10_SafetyGate7_DB"."sSafetyGate UnlockRequest" := FALSE;
       "ST10_SafetyGate7_DB"."sSafetyGate LockRequest" := TRUE;
       "ST10_SafetyGate_InterfaceDB".J.Status_3 := 4;
   END_IF;
   IF #_w1 AND ("ST10_SafetyGate_InterfaceDB".J.Status_3 <> 1) AND ("ST10_SafetyGate_InterfaceDB".J.Status_3 <> 2) AND ("ST10_SafetyGate_InterfaceDB".J.Status_3 <> 3) AND ("ST10_SafetyGate_InterfaceDB".J.Status_3 <> 4) THEN
       "ST10_SafetyGate_InterfaceDB".J.Status_3 := 1;
   END_IF;
   IF #_w1 AND ("ST10_SafetyGate_InterfaceDB".J.Status_3 = 2) AND NOT "iMagnet_UnlockButton" THEN
       "ST10_SafetyGate_InterfaceDB".J.Status_3 := 3;
   END_IF;
   IF #_w1 AND ("ST10_SafetyGate_InterfaceDB".J.Status_3 = 4) AND NOT "iMagnet_UnlockButton" THEN
       "ST10_SafetyGate_InterfaceDB".J.Status_3 := 5;
   END_IF;
END_REGION

REGION Network 23: E-NG料盒-02安全门锁按钮灯
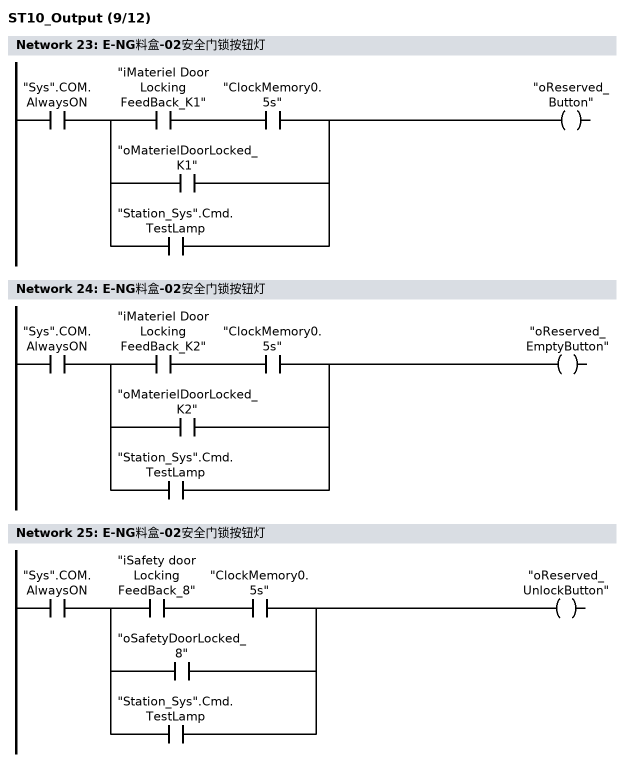
   RUNG wire#powerrail
      Contact( "Sys".COM.AlwaysON )
      wire#w1
      Contact( "iMateriel Door Locking FeedBack_K1" )
      Contact( "ClockMemory0.5s" )
      wire#w2
      Coil( "oReserved_Button" )
   END_RUNG
   RUNG wire#w1
      Contact( "oMaterielDoorLocked_K1" )
   END_RUNG wire#w2
   RUNG wire#w1
      Contact( "Station_Sys".Cmd.TestLamp )
   END_RUNG wire#w2
   // the same network as SCL:
   "oReserved_Button" := "Sys".COM.AlwaysON AND (("iMateriel Door Locking FeedBack_K1" AND "ClockMemory0.5s") OR "oMaterielDoorLocked_K1" OR "Station_Sys".Cmd.TestLamp);
END_REGION

REGION Network 24: E-NG料盒-02安全门锁按钮灯
   RUNG wire#powerrail
      Contact( "Sys".COM.AlwaysON )
      wire#w1
      Contact( "iMateriel Door Locking FeedBack_K2" )
      Contact( "ClockMemory0.5s" )
      wire#w2
      Coil( "oReserved_EmptyButton" )
   END_RUNG
   RUNG wire#w1
      Contact( "oMaterielDoorLocked_K2" )
   END_RUNG wire#w2
   RUNG wire#w1
      Contact( "Station_Sys".Cmd.TestLamp )
   END_RUNG wire#w2
   // the same network as SCL:
   "oReserved_EmptyButton" := "Sys".COM.AlwaysON AND (("iMateriel Door Locking FeedBack_K2" AND "ClockMemory0.5s") OR "oMaterielDoorLocked_K2" OR "Station_Sys".Cmd.TestLamp);
END_REGION

REGION Network 25: E-NG料盒-02安全门锁按钮灯
   RUNG wire#powerrail
      Contact( "Sys".COM.AlwaysON )
      wire#w1
      Contact( "iSafety door Locking FeedBack_8" )
      Contact( "ClockMemory0.5s" )
      wire#w2
      Coil( "oReserved_UnlockButton" )
   END_RUNG
   RUNG wire#w1
      Contact( "oSafetyDoorLocked_8" )
   END_RUNG wire#w2
   RUNG wire#w1
      Contact( "Station_Sys".Cmd.TestLamp )
   END_RUNG wire#w2
   // the same network as SCL:
   "oReserved_UnlockButton" := "Sys".COM.AlwaysON AND (("iSafety door Locking FeedBack_8" AND "ClockMemory0.5s") OR "oSafetyDoorLocked_8" OR "Station_Sys".Cmd.TestLamp);
END_REGION

REGION Network 26
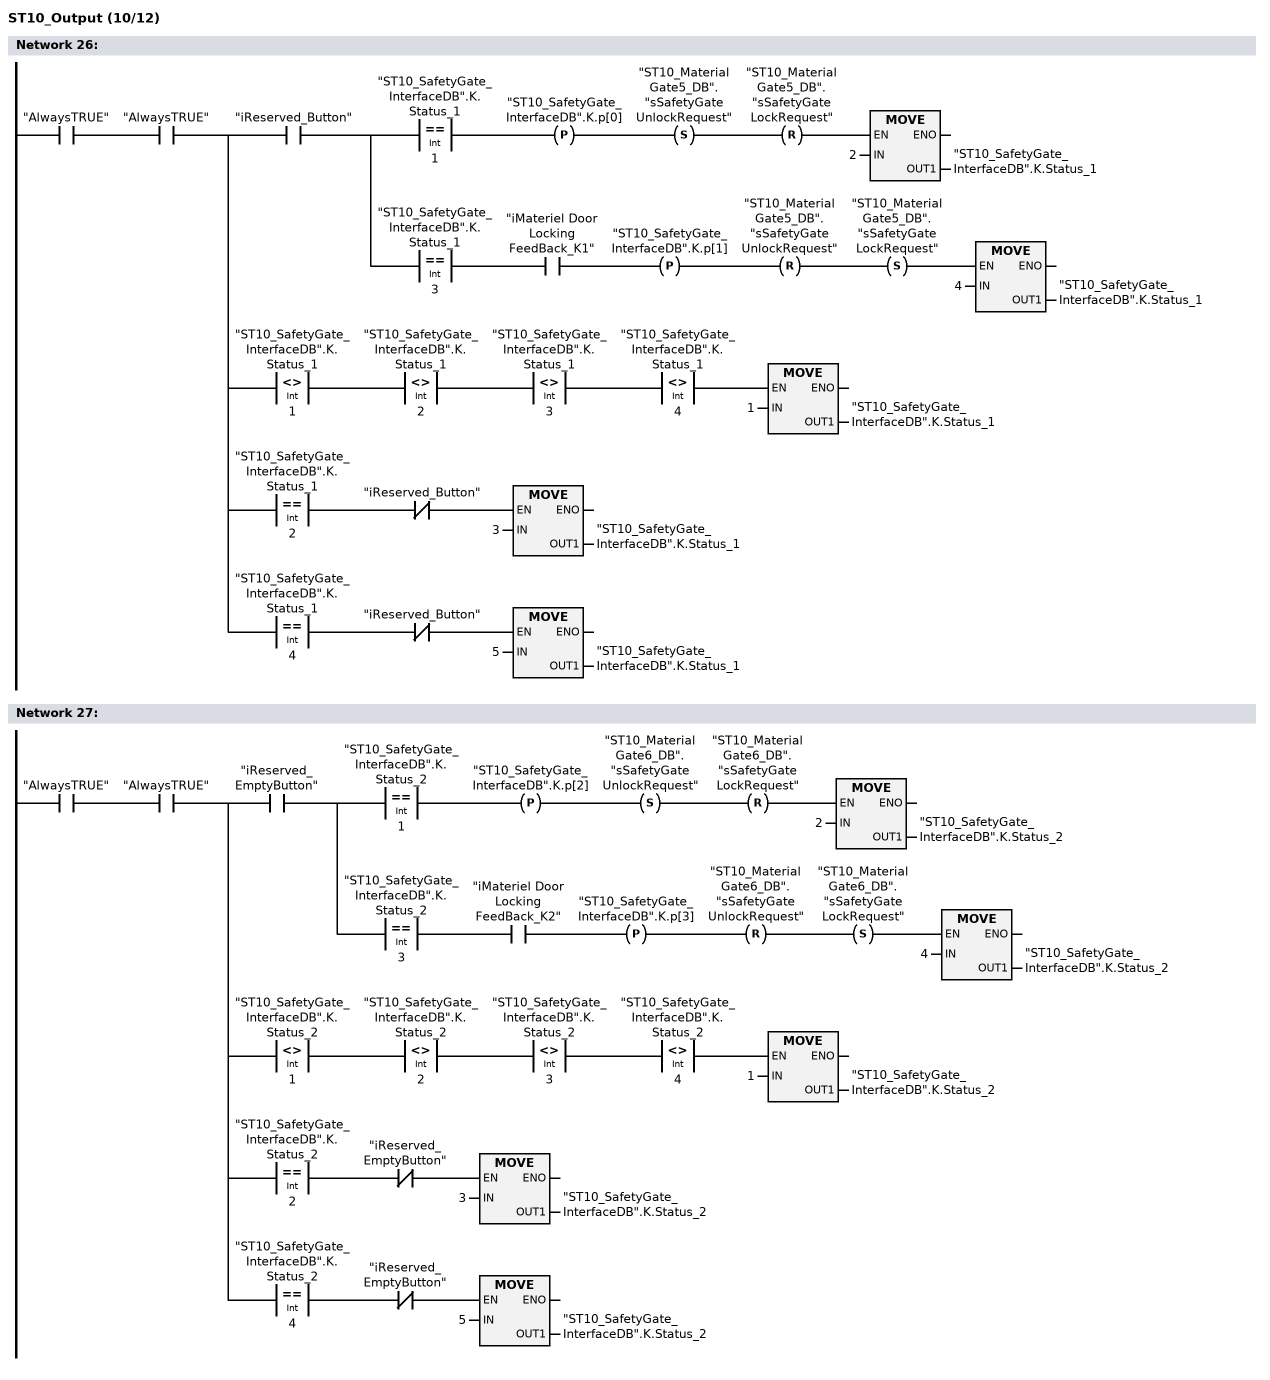
   RUNG wire#powerrail
      Contact( "AlwaysTRUE" )
      Contact( "AlwaysTRUE" )
      wire#w1
      Contact( "iReserved_Button" )
      wire#w2
      { S7_Templates := "SrcType := Int" } EQ_Contact(in1 := "ST10_SafetyGate_InterfaceDB".K.Status_1, in2 := 1)
      P_Trig( "ST10_SafetyGate_InterfaceDB".K.p[0] )
      S_Coil( "ST10_MaterialGate5_DB"."sSafetyGate UnlockRequest" )
      R_Coil( "ST10_MaterialGate5_DB"."sSafetyGate LockRequest" )
      Move(in := 2, out1 => "ST10_SafetyGate_InterfaceDB".K.Status_1)
   END_RUNG
   RUNG wire#w2
      { S7_Templates := "SrcType := Int" } EQ_Contact(in1 := "ST10_SafetyGate_InterfaceDB".K.Status_1, in2 := 3)
      Contact( "iMateriel Door Locking FeedBack_K1" )
      P_Trig( "ST10_SafetyGate_InterfaceDB".K.p[1] )
      R_Coil( "ST10_MaterialGate5_DB"."sSafetyGate UnlockRequest" )
      S_Coil( "ST10_MaterialGate5_DB"."sSafetyGate LockRequest" )
      Move(in := 4, out1 => "ST10_SafetyGate_InterfaceDB".K.Status_1)
   END_RUNG
   RUNG wire#w1
      { S7_Templates := "SrcType := Int" } NE_Contact(in1 := "ST10_SafetyGate_InterfaceDB".K.Status_1, in2 := 1)
      { S7_Templates := "SrcType := Int" } NE_Contact(in1 := "ST10_SafetyGate_InterfaceDB".K.Status_1, in2 := 2)
      { S7_Templates := "SrcType := Int" } NE_Contact(in1 := "ST10_SafetyGate_InterfaceDB".K.Status_1, in2 := 3)
      { S7_Templates := "SrcType := Int" } NE_Contact(in1 := "ST10_SafetyGate_InterfaceDB".K.Status_1, in2 := 4)
      Move(in := 1, out1 => "ST10_SafetyGate_InterfaceDB".K.Status_1)
   END_RUNG
   RUNG wire#w1
      { S7_Templates := "SrcType := Int" } EQ_Contact(in1 := "ST10_SafetyGate_InterfaceDB".K.Status_1, in2 := 2)
      I_Contact( "iReserved_Button" )
      Move(in := 3, out1 => "ST10_SafetyGate_InterfaceDB".K.Status_1)
   END_RUNG
   RUNG wire#w1
      { S7_Templates := "SrcType := Int" } EQ_Contact(in1 := "ST10_SafetyGate_InterfaceDB".K.Status_1, in2 := 4)
      I_Contact( "iReserved_Button" )
      Move(in := 5, out1 => "ST10_SafetyGate_InterfaceDB".K.Status_1)
   END_RUNG
   // the same network as SCL:
   #_w1 := "AlwaysTRUE" AND "AlwaysTRUE";
   #_w2 := #_w1 AND "iReserved_Button";
   #_w3 := #_w2 AND ("ST10_SafetyGate_InterfaceDB".K.Status_1 = 1);
   #_w4 := #_w3 AND NOT "ST10_SafetyGate_InterfaceDB".K.p[0];   // rising edge
   "ST10_SafetyGate_InterfaceDB".K.p[0] := #_w3;
   IF #_w4 THEN
       "ST10_MaterialGate5_DB"."sSafetyGate UnlockRequest" := TRUE;
       "ST10_MaterialGate5_DB"."sSafetyGate LockRequest" := FALSE;
       "ST10_SafetyGate_InterfaceDB".K.Status_1 := 2;
   END_IF;
   #_w5 := #_w2 AND ("ST10_SafetyGate_InterfaceDB".K.Status_1 = 3) AND "iMateriel Door Locking FeedBack_K1";
   #_w6 := #_w5 AND NOT "ST10_SafetyGate_InterfaceDB".K.p[1];   // rising edge
   "ST10_SafetyGate_InterfaceDB".K.p[1] := #_w5;
   IF #_w6 THEN
       "ST10_MaterialGate5_DB"."sSafetyGate UnlockRequest" := FALSE;
       "ST10_MaterialGate5_DB"."sSafetyGate LockRequest" := TRUE;
       "ST10_SafetyGate_InterfaceDB".K.Status_1 := 4;
   END_IF;
   IF #_w1 AND ("ST10_SafetyGate_InterfaceDB".K.Status_1 <> 1) AND ("ST10_SafetyGate_InterfaceDB".K.Status_1 <> 2) AND ("ST10_SafetyGate_InterfaceDB".K.Status_1 <> 3) AND ("ST10_SafetyGate_InterfaceDB".K.Status_1 <> 4) THEN
       "ST10_SafetyGate_InterfaceDB".K.Status_1 := 1;
   END_IF;
   IF #_w1 AND ("ST10_SafetyGate_InterfaceDB".K.Status_1 = 2) AND NOT "iReserved_Button" THEN
       "ST10_SafetyGate_InterfaceDB".K.Status_1 := 3;
   END_IF;
   IF #_w1 AND ("ST10_SafetyGate_InterfaceDB".K.Status_1 = 4) AND NOT "iReserved_Button" THEN
       "ST10_SafetyGate_InterfaceDB".K.Status_1 := 5;
   END_IF;
END_REGION

REGION Network 27
   RUNG wire#powerrail
      Contact( "AlwaysTRUE" )
      Contact( "AlwaysTRUE" )
      wire#w1
      Contact( "iReserved_EmptyButton" )
      wire#w2
      { S7_Templates := "SrcType := Int" } EQ_Contact(in1 := "ST10_SafetyGate_InterfaceDB".K.Status_2, in2 := 1)
      P_Trig( "ST10_SafetyGate_InterfaceDB".K.p[2] )
      S_Coil( "ST10_MaterialGate6_DB"."sSafetyGate UnlockRequest" )
      R_Coil( "ST10_MaterialGate6_DB"."sSafetyGate LockRequest" )
      Move(in := 2, out1 => "ST10_SafetyGate_InterfaceDB".K.Status_2)
   END_RUNG
   RUNG wire#w2
      { S7_Templates := "SrcType := Int" } EQ_Contact(in1 := "ST10_SafetyGate_InterfaceDB".K.Status_2, in2 := 3)
      Contact( "iMateriel Door Locking FeedBack_K2" )
      P_Trig( "ST10_SafetyGate_InterfaceDB".K.p[3] )
      R_Coil( "ST10_MaterialGate6_DB"."sSafetyGate UnlockRequest" )
      S_Coil( "ST10_MaterialGate6_DB"."sSafetyGate LockRequest" )
      Move(in := 4, out1 => "ST10_SafetyGate_InterfaceDB".K.Status_2)
   END_RUNG
   RUNG wire#w1
      { S7_Templates := "SrcType := Int" } NE_Contact(in1 := "ST10_SafetyGate_InterfaceDB".K.Status_2, in2 := 1)
      { S7_Templates := "SrcType := Int" } NE_Contact(in1 := "ST10_SafetyGate_InterfaceDB".K.Status_2, in2 := 2)
      { S7_Templates := "SrcType := Int" } NE_Contact(in1 := "ST10_SafetyGate_InterfaceDB".K.Status_2, in2 := 3)
      { S7_Templates := "SrcType := Int" } NE_Contact(in1 := "ST10_SafetyGate_InterfaceDB".K.Status_2, in2 := 4)
      Move(in := 1, out1 => "ST10_SafetyGate_InterfaceDB".K.Status_2)
   END_RUNG
   RUNG wire#w1
      { S7_Templates := "SrcType := Int" } EQ_Contact(in1 := "ST10_SafetyGate_InterfaceDB".K.Status_2, in2 := 2)
      I_Contact( "iReserved_EmptyButton" )
      Move(in := 3, out1 => "ST10_SafetyGate_InterfaceDB".K.Status_2)
   END_RUNG
   RUNG wire#w1
      { S7_Templates := "SrcType := Int" } EQ_Contact(in1 := "ST10_SafetyGate_InterfaceDB".K.Status_2, in2 := 4)
      I_Contact( "iReserved_EmptyButton" )
      Move(in := 5, out1 => "ST10_SafetyGate_InterfaceDB".K.Status_2)
   END_RUNG
   // the same network as SCL:
   #_w1 := "AlwaysTRUE" AND "AlwaysTRUE";
   #_w2 := #_w1 AND "iReserved_EmptyButton";
   #_w3 := #_w2 AND ("ST10_SafetyGate_InterfaceDB".K.Status_2 = 1);
   #_w4 := #_w3 AND NOT "ST10_SafetyGate_InterfaceDB".K.p[2];   // rising edge
   "ST10_SafetyGate_InterfaceDB".K.p[2] := #_w3;
   IF #_w4 THEN
       "ST10_MaterialGate6_DB"."sSafetyGate UnlockRequest" := TRUE;
       "ST10_MaterialGate6_DB"."sSafetyGate LockRequest" := FALSE;
       "ST10_SafetyGate_InterfaceDB".K.Status_2 := 2;
   END_IF;
   #_w5 := #_w2 AND ("ST10_SafetyGate_InterfaceDB".K.Status_2 = 3) AND "iMateriel Door Locking FeedBack_K2";
   #_w6 := #_w5 AND NOT "ST10_SafetyGate_InterfaceDB".K.p[3];   // rising edge
   "ST10_SafetyGate_InterfaceDB".K.p[3] := #_w5;
   IF #_w6 THEN
       "ST10_MaterialGate6_DB"."sSafetyGate UnlockRequest" := FALSE;
       "ST10_MaterialGate6_DB"."sSafetyGate LockRequest" := TRUE;
       "ST10_SafetyGate_InterfaceDB".K.Status_2 := 4;
   END_IF;
   IF #_w1 AND ("ST10_SafetyGate_InterfaceDB".K.Status_2 <> 1) AND ("ST10_SafetyGate_InterfaceDB".K.Status_2 <> 2) AND ("ST10_SafetyGate_InterfaceDB".K.Status_2 <> 3) AND ("ST10_SafetyGate_InterfaceDB".K.Status_2 <> 4) THEN
       "ST10_SafetyGate_InterfaceDB".K.Status_2 := 1;
   END_IF;
   IF #_w1 AND ("ST10_SafetyGate_InterfaceDB".K.Status_2 = 2) AND NOT "iReserved_EmptyButton" THEN
       "ST10_SafetyGate_InterfaceDB".K.Status_2 := 3;
   END_IF;
   IF #_w1 AND ("ST10_SafetyGate_InterfaceDB".K.Status_2 = 4) AND NOT "iReserved_EmptyButton" THEN
       "ST10_SafetyGate_InterfaceDB".K.Status_2 := 5;
   END_IF;
END_REGION

REGION Network 28
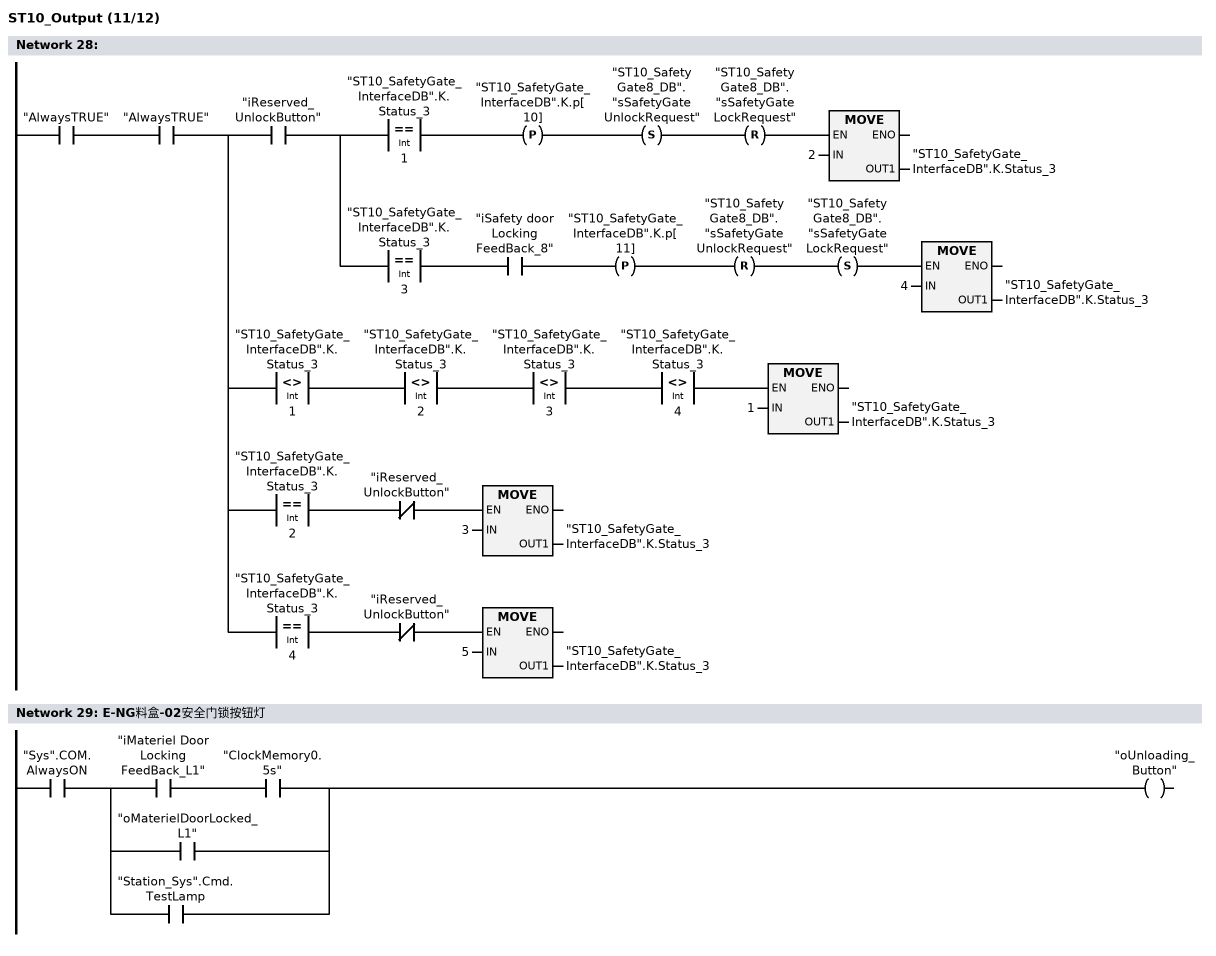
   RUNG wire#powerrail
      Contact( "AlwaysTRUE" )
      Contact( "AlwaysTRUE" )
      wire#w1
      Contact( "iReserved_UnlockButton" )
      wire#w2
      { S7_Templates := "SrcType := Int" } EQ_Contact(in1 := "ST10_SafetyGate_InterfaceDB".K.Status_3, in2 := 1)
      P_Trig( "ST10_SafetyGate_InterfaceDB".K.p[10] )
      S_Coil( "ST10_SafetyGate8_DB"."sSafetyGate UnlockRequest" )
      R_Coil( "ST10_SafetyGate8_DB"."sSafetyGate LockRequest" )
      Move(in := 2, out1 => "ST10_SafetyGate_InterfaceDB".K.Status_3)
   END_RUNG
   RUNG wire#w2
      { S7_Templates := "SrcType := Int" } EQ_Contact(in1 := "ST10_SafetyGate_InterfaceDB".K.Status_3, in2 := 3)
      Contact( "iSafety door Locking FeedBack_8" )
      P_Trig( "ST10_SafetyGate_InterfaceDB".K.p[11] )
      R_Coil( "ST10_SafetyGate8_DB"."sSafetyGate UnlockRequest" )
      S_Coil( "ST10_SafetyGate8_DB"."sSafetyGate LockRequest" )
      Move(in := 4, out1 => "ST10_SafetyGate_InterfaceDB".K.Status_3)
   END_RUNG
   RUNG wire#w1
      { S7_Templates := "SrcType := Int" } NE_Contact(in1 := "ST10_SafetyGate_InterfaceDB".K.Status_3, in2 := 1)
      { S7_Templates := "SrcType := Int" } NE_Contact(in1 := "ST10_SafetyGate_InterfaceDB".K.Status_3, in2 := 2)
      { S7_Templates := "SrcType := Int" } NE_Contact(in1 := "ST10_SafetyGate_InterfaceDB".K.Status_3, in2 := 3)
      { S7_Templates := "SrcType := Int" } NE_Contact(in1 := "ST10_SafetyGate_InterfaceDB".K.Status_3, in2 := 4)
      Move(in := 1, out1 => "ST10_SafetyGate_InterfaceDB".K.Status_3)
   END_RUNG
   RUNG wire#w1
      { S7_Templates := "SrcType := Int" } EQ_Contact(in1 := "ST10_SafetyGate_InterfaceDB".K.Status_3, in2 := 2)
      I_Contact( "iReserved_UnlockButton" )
      Move(in := 3, out1 => "ST10_SafetyGate_InterfaceDB".K.Status_3)
   END_RUNG
   RUNG wire#w1
      { S7_Templates := "SrcType := Int" } EQ_Contact(in1 := "ST10_SafetyGate_InterfaceDB".K.Status_3, in2 := 4)
      I_Contact( "iReserved_UnlockButton" )
      Move(in := 5, out1 => "ST10_SafetyGate_InterfaceDB".K.Status_3)
   END_RUNG
   // the same network as SCL:
   #_w1 := "AlwaysTRUE" AND "AlwaysTRUE";
   #_w2 := #_w1 AND "iReserved_UnlockButton";
   #_w3 := #_w2 AND ("ST10_SafetyGate_InterfaceDB".K.Status_3 = 1);
   #_w4 := #_w3 AND NOT "ST10_SafetyGate_InterfaceDB".K.p[10];   // rising edge
   "ST10_SafetyGate_InterfaceDB".K.p[10] := #_w3;
   IF #_w4 THEN
       "ST10_SafetyGate8_DB"."sSafetyGate UnlockRequest" := TRUE;
       "ST10_SafetyGate8_DB"."sSafetyGate LockRequest" := FALSE;
       "ST10_SafetyGate_InterfaceDB".K.Status_3 := 2;
   END_IF;
   #_w5 := #_w2 AND ("ST10_SafetyGate_InterfaceDB".K.Status_3 = 3) AND "iSafety door Locking FeedBack_8";
   #_w6 := #_w5 AND NOT "ST10_SafetyGate_InterfaceDB".K.p[11];   // rising edge
   "ST10_SafetyGate_InterfaceDB".K.p[11] := #_w5;
   IF #_w6 THEN
       "ST10_SafetyGate8_DB"."sSafetyGate UnlockRequest" := FALSE;
       "ST10_SafetyGate8_DB"."sSafetyGate LockRequest" := TRUE;
       "ST10_SafetyGate_InterfaceDB".K.Status_3 := 4;
   END_IF;
   IF #_w1 AND ("ST10_SafetyGate_InterfaceDB".K.Status_3 <> 1) AND ("ST10_SafetyGate_InterfaceDB".K.Status_3 <> 2) AND ("ST10_SafetyGate_InterfaceDB".K.Status_3 <> 3) AND ("ST10_SafetyGate_InterfaceDB".K.Status_3 <> 4) THEN
       "ST10_SafetyGate_InterfaceDB".K.Status_3 := 1;
   END_IF;
   IF #_w1 AND ("ST10_SafetyGate_InterfaceDB".K.Status_3 = 2) AND NOT "iReserved_UnlockButton" THEN
       "ST10_SafetyGate_InterfaceDB".K.Status_3 := 3;
   END_IF;
   IF #_w1 AND ("ST10_SafetyGate_InterfaceDB".K.Status_3 = 4) AND NOT "iReserved_UnlockButton" THEN
       "ST10_SafetyGate_InterfaceDB".K.Status_3 := 5;
   END_IF;
END_REGION

REGION Network 29: E-NG料盒-02安全门锁按钮灯
   RUNG wire#powerrail
      Contact( "Sys".COM.AlwaysON )
      wire#w1
      Contact( "iMateriel Door Locking FeedBack_L1" )
      Contact( "ClockMemory0.5s" )
      wire#w2
      Coil( "oUnloading_Button" )
   END_RUNG
   RUNG wire#w1
      Contact( "oMaterielDoorLocked_L1" )
   END_RUNG wire#w2
   RUNG wire#w1
      Contact( "Station_Sys".Cmd.TestLamp )
   END_RUNG wire#w2
   // the same network as SCL:
   "oUnloading_Button" := "Sys".COM.AlwaysON AND (("iMateriel Door Locking FeedBack_L1" AND "ClockMemory0.5s") OR "oMaterielDoorLocked_L1" OR "Station_Sys".Cmd.TestLamp);
END_REGION

REGION Network 30
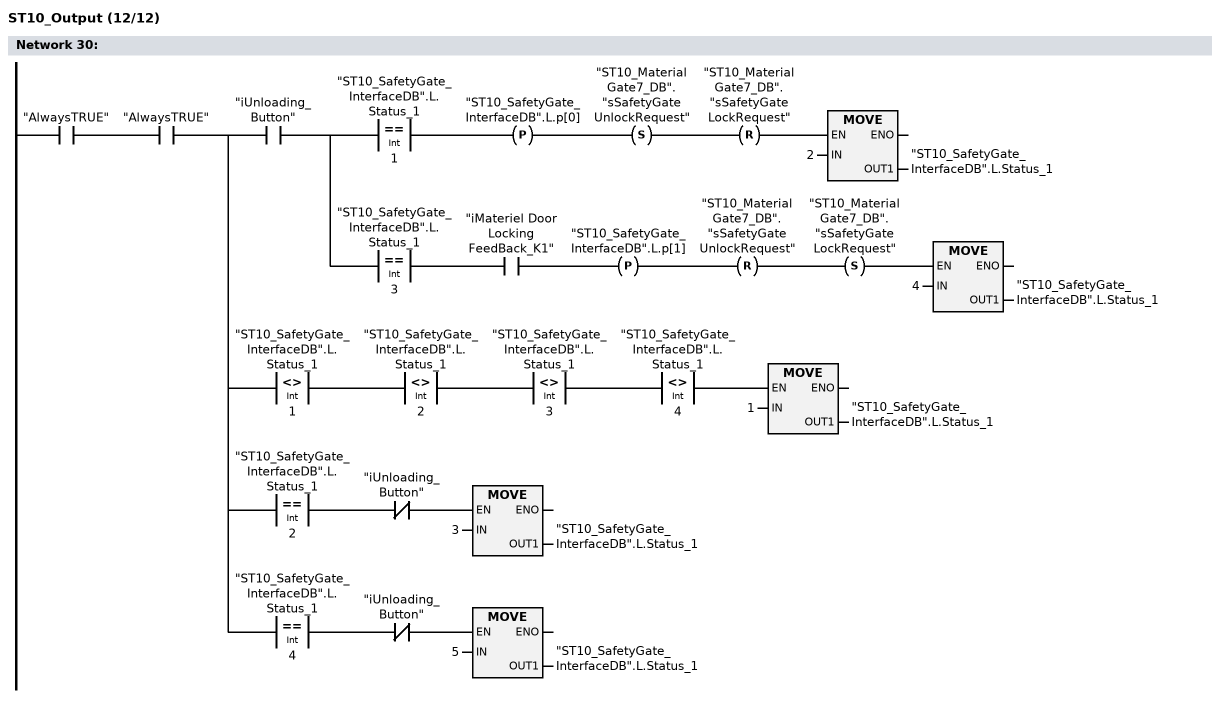
   RUNG wire#powerrail
      Contact( "AlwaysTRUE" )
      Contact( "AlwaysTRUE" )
      wire#w1
      Contact( "iUnloading_Button" )
      wire#w2
      { S7_Templates := "SrcType := Int" } EQ_Contact(in1 := "ST10_SafetyGate_InterfaceDB".L.Status_1, in2 := 1)
      P_Trig( "ST10_SafetyGate_InterfaceDB".L.p[0] )
      S_Coil( "ST10_MaterialGate7_DB"."sSafetyGate UnlockRequest" )
      R_Coil( "ST10_MaterialGate7_DB"."sSafetyGate LockRequest" )
      Move(in := 2, out1 => "ST10_SafetyGate_InterfaceDB".L.Status_1)
   END_RUNG
   RUNG wire#w2
      { S7_Templates := "SrcType := Int" } EQ_Contact(in1 := "ST10_SafetyGate_InterfaceDB".L.Status_1, in2 := 3)
      Contact( "iMateriel Door Locking FeedBack_K1" )
      P_Trig( "ST10_SafetyGate_InterfaceDB".L.p[1] )
      R_Coil( "ST10_MaterialGate7_DB"."sSafetyGate UnlockRequest" )
      S_Coil( "ST10_MaterialGate7_DB"."sSafetyGate LockRequest" )
      Move(in := 4, out1 => "ST10_SafetyGate_InterfaceDB".L.Status_1)
   END_RUNG
   RUNG wire#w1
      { S7_Templates := "SrcType := Int" } NE_Contact(in1 := "ST10_SafetyGate_InterfaceDB".L.Status_1, in2 := 1)
      { S7_Templates := "SrcType := Int" } NE_Contact(in1 := "ST10_SafetyGate_InterfaceDB".L.Status_1, in2 := 2)
      { S7_Templates := "SrcType := Int" } NE_Contact(in1 := "ST10_SafetyGate_InterfaceDB".L.Status_1, in2 := 3)
      { S7_Templates := "SrcType := Int" } NE_Contact(in1 := "ST10_SafetyGate_InterfaceDB".L.Status_1, in2 := 4)
      Move(in := 1, out1 => "ST10_SafetyGate_InterfaceDB".L.Status_1)
   END_RUNG
   RUNG wire#w1
      { S7_Templates := "SrcType := Int" } EQ_Contact(in1 := "ST10_SafetyGate_InterfaceDB".L.Status_1, in2 := 2)
      I_Contact( "iUnloading_Button" )
      Move(in := 3, out1 => "ST10_SafetyGate_InterfaceDB".L.Status_1)
   END_RUNG
   RUNG wire#w1
      { S7_Templates := "SrcType := Int" } EQ_Contact(in1 := "ST10_SafetyGate_InterfaceDB".L.Status_1, in2 := 4)
      I_Contact( "iUnloading_Button" )
      Move(in := 5, out1 => "ST10_SafetyGate_InterfaceDB".L.Status_1)
   END_RUNG
   // the same network as SCL:
   #_w1 := "AlwaysTRUE" AND "AlwaysTRUE";
   #_w2 := #_w1 AND "iUnloading_Button";
   #_w3 := #_w2 AND ("ST10_SafetyGate_InterfaceDB".L.Status_1 = 1);
   #_w4 := #_w3 AND NOT "ST10_SafetyGate_InterfaceDB".L.p[0];   // rising edge
   "ST10_SafetyGate_InterfaceDB".L.p[0] := #_w3;
   IF #_w4 THEN
       "ST10_MaterialGate7_DB"."sSafetyGate UnlockRequest" := TRUE;
       "ST10_MaterialGate7_DB"."sSafetyGate LockRequest" := FALSE;
       "ST10_SafetyGate_InterfaceDB".L.Status_1 := 2;
   END_IF;
   #_w5 := #_w2 AND ("ST10_SafetyGate_InterfaceDB".L.Status_1 = 3) AND "iMateriel Door Locking FeedBack_K1";
   #_w6 := #_w5 AND NOT "ST10_SafetyGate_InterfaceDB".L.p[1];   // rising edge
   "ST10_SafetyGate_InterfaceDB".L.p[1] := #_w5;
   IF #_w6 THEN
       "ST10_MaterialGate7_DB"."sSafetyGate UnlockRequest" := FALSE;
       "ST10_MaterialGate7_DB"."sSafetyGate LockRequest" := TRUE;
       "ST10_SafetyGate_InterfaceDB".L.Status_1 := 4;
   END_IF;
   IF #_w1 AND ("ST10_SafetyGate_InterfaceDB".L.Status_1 <> 1) AND ("ST10_SafetyGate_InterfaceDB".L.Status_1 <> 2) AND ("ST10_SafetyGate_InterfaceDB".L.Status_1 <> 3) AND ("ST10_SafetyGate_InterfaceDB".L.Status_1 <> 4) THEN
       "ST10_SafetyGate_InterfaceDB".L.Status_1 := 1;
   END_IF;
   IF #_w1 AND ("ST10_SafetyGate_InterfaceDB".L.Status_1 = 2) AND NOT "iUnloading_Button" THEN
       "ST10_SafetyGate_InterfaceDB".L.Status_1 := 3;
   END_IF;
   IF #_w1 AND ("ST10_SafetyGate_InterfaceDB".L.Status_1 = 4) AND NOT "iUnloading_Button" THEN
       "ST10_SafetyGate_InterfaceDB".L.Status_1 := 5;
   END_IF;
END_REGION
END_FUNCTION

FUNCTION_BLOCK "FB_Tower_4Lamp"   // FB5050, LAD
{ S7_Optimized_Access := 'TRUE' }
VERSION : 0.1
// stored: AutoNumber false, IsIECCheckEnabled false, IsRetainMemResEnabled false, MemoryReserve 100, SetENOAutomatically false, UDAEnableTagReadback false
   VAR_INPUT
      iReady : Bool;   // 系统OK
      iManual_Mode : Bool;
      iAuto_Mode : Bool;
      iAuto_Running : Bool;   // 自动运行信号
      iCheck_Mode : Bool;
      iIdle : Bool;   // 自动运行中空闲信号
      iWarning : Bool;
      iFault : Bool;
      "i0.5s_Pulse" : Bool;   // 0.5S脉冲
      i1s_Pulse : Bool;   // 1S脉冲
      i2s_Pulse : Bool;   // 2S脉冲
      iResetButton : Bool;   // 复位按钮
      "iE-StopButtonOK" : Bool;   // 急停按钮未按下
      iSafetyGateClosed : Bool;   // 安全门关闭信号
      iSafetyGateRelayOK : Bool;   // 安全门继电器输出OK
      iPowerOn : Bool;   // 系统上电信号
      iMachineHomePos : Bool;   // 所有设备在原始位
      iWorkAreaLightButton : Bool;   // HMI工作区域照明按钮
      iTest_Lamp : Bool;   // 灯测试按钮
   END_VAR
   VAR_OUTPUT
      oRed_Lamp : Bool;   // 塔灯-红色
      oYellow_Lamp : Bool;   // 塔灯-黄色
      oGreen_Lamp : Bool;   // 塔灯-绿色
      oBlue_Lamp : Bool;   // 塔灯-蓝色 1.蓝灯常亮表示设备在原位;2.蓝灯闪烁表示工位缺料等待上料
      oBuzzer : Bool;   // 塔灯-蜂鸣器
      oPowerOn : Bool;   // 系统上电指示灯
      oResetLamp : Bool;   // 复位按钮指示灯
      oWorkArea1_LightingOn : Bool;   // 工作区域1 照明打开
      oWorkArea2_LightingOn : Bool;   // 工作区域2 照明打开
      oWorkArea3_LightingOn : Bool;   // 工作区域3 照明打开
   END_VAR
   VAR_IN_OUT
      ioStationWaitingLoadPart : Bool;   // 工位等待工位上料
      ioBuzzerON : Bool;   // 蜂鸣器屏蔽开关
      ioBuzzerSetVal : Int;   // 蜂鸣器鸣叫设定值
   END_VAR
   VAR
      TON : Array[0..10] of TON_TIME;
      sRed_Lamp { S7_SetPoint := 'True'} : Bool;
      sResetButtonPressed : Bool;   // 复位按钮已按下
      sBuzzerOnCurrentVal : Int;   // 蜂鸣器鸣叫实际值
      P_TRIG : Array[0..10] of Bool;
      N_TRIG : Array[0..10] of Bool;
   END_VAR
   VAR_TEMP   // added for the SCL form of the ladder/FBD networks
      _w1 : Bool;
      _w2 : Bool;
      _w3 : Bool;
      _w4 : Bool;
      _w5 : Bool;
      _w6 : Bool;
   END_VAR
BEGIN

REGION Network 1: 塔灯-红色 / TowerLamp_Red
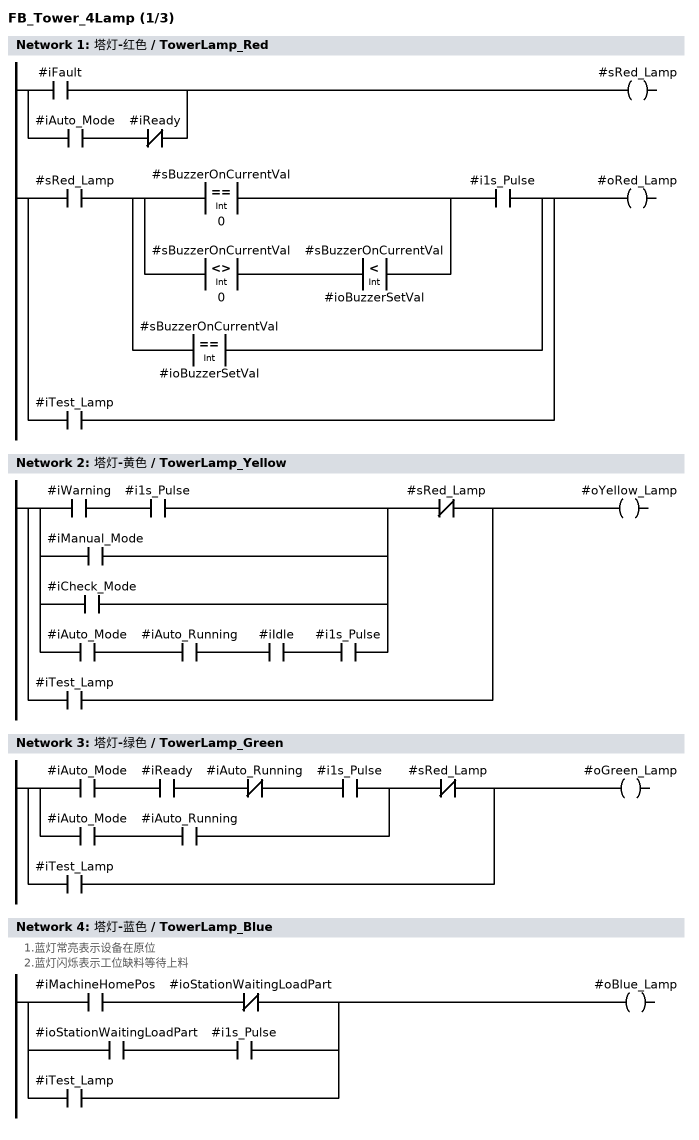
   RUNG wire#powerrail
      Contact( #iFault )
      wire#w1
      Coil( #sRed_Lamp )
   END_RUNG
   RUNG wire#powerrail
      Contact( #iAuto_Mode )
      I_Contact( #iReady )
   END_RUNG wire#w1
   RUNG wire#powerrail
      Contact( #sRed_Lamp )
      wire#w2
      { S7_Templates := "SrcType := Int" } EQ_Contact(in1 := #sBuzzerOnCurrentVal, in2 := 0)
      wire#w3
      Contact( #i1s_Pulse )
      wire#w4
      Coil( #oRed_Lamp )
   END_RUNG
   RUNG wire#w2
      { S7_Templates := "SrcType := Int" } NE_Contact(in1 := #sBuzzerOnCurrentVal, in2 := 0)
      { S7_Templates := "SrcType := Int" } LT_Contact(in1 := #sBuzzerOnCurrentVal, in2 := #ioBuzzerSetVal)
   END_RUNG wire#w3
   RUNG wire#w2
      { S7_Templates := "SrcType := Int" } EQ_Contact(in1 := #sBuzzerOnCurrentVal, in2 := #ioBuzzerSetVal)
   END_RUNG wire#w4
   RUNG wire#powerrail
      Contact( #iTest_Lamp )
   END_RUNG wire#w4
   // the same network as SCL:
   #sRed_Lamp := #iFault OR (#iAuto_Mode AND NOT #iReady);
   #oRed_Lamp := (#sRed_Lamp AND ((((#sBuzzerOnCurrentVal = 0) OR ((#sBuzzerOnCurrentVal <> 0) AND (#sBuzzerOnCurrentVal < #ioBuzzerSetVal))) AND #i1s_Pulse) OR (#sBuzzerOnCurrentVal = #ioBuzzerSetVal))) OR #iTest_Lamp;
END_REGION

REGION Network 2: 塔灯-黄色 / TowerLamp_Yellow
   RUNG wire#powerrail
      Contact( #iWarning )
      Contact( #i1s_Pulse )
      wire#w1
      I_Contact( #sRed_Lamp )
      wire#w2
      Coil( #oYellow_Lamp )
   END_RUNG
   RUNG wire#powerrail
      Contact( #iManual_Mode )
   END_RUNG wire#w1
   RUNG wire#powerrail
      Contact( #iCheck_Mode )
   END_RUNG wire#w1
   RUNG wire#powerrail
      Contact( #iAuto_Mode )
      Contact( #iAuto_Running )
      Contact( #iIdle )
      Contact( #i1s_Pulse )
   END_RUNG wire#w1
   RUNG wire#powerrail
      Contact( #iTest_Lamp )
   END_RUNG wire#w2
   // the same network as SCL:
   #oYellow_Lamp := (((#iWarning AND #i1s_Pulse) OR #iManual_Mode OR #iCheck_Mode OR (#iAuto_Mode AND #iAuto_Running AND #iIdle AND #i1s_Pulse)) AND NOT #sRed_Lamp) OR #iTest_Lamp;
END_REGION

REGION Network 3: 塔灯-绿色 / TowerLamp_Green
   RUNG wire#powerrail
      Contact( #iAuto_Mode )
      Contact( #iReady )
      I_Contact( #iAuto_Running )
      Contact( #i1s_Pulse )
      wire#w1
      I_Contact( #sRed_Lamp )
      wire#w2
      Coil( #oGreen_Lamp )
   END_RUNG
   RUNG wire#powerrail
      Contact( #iAuto_Mode )
      Contact( #iAuto_Running )
   END_RUNG wire#w1
   RUNG wire#powerrail
      Contact( #iTest_Lamp )
   END_RUNG wire#w2
   // the same network as SCL:
   #oGreen_Lamp := (((#iAuto_Mode AND #iReady AND NOT #iAuto_Running AND #i1s_Pulse) OR (#iAuto_Mode AND #iAuto_Running)) AND NOT #sRed_Lamp) OR #iTest_Lamp;
END_REGION

REGION Network 4: 塔灯-蓝色 / TowerLamp_Blue
   // 1.蓝灯常亮表示设备在原位
   // 2.蓝灯闪烁表示工位缺料等待上料
   RUNG wire#powerrail
      Contact( #iMachineHomePos )
      I_Contact( #ioStationWaitingLoadPart )
      wire#w1
      Coil( #oBlue_Lamp )
   END_RUNG
   RUNG wire#powerrail
      Contact( #ioStationWaitingLoadPart )
      Contact( #i1s_Pulse )
   END_RUNG wire#w1
   RUNG wire#powerrail
      Contact( #iTest_Lamp )
   END_RUNG wire#w1
   // the same network as SCL:
   #oBlue_Lamp := (#iMachineHomePos AND NOT #ioStationWaitingLoadPart) OR (#ioStationWaitingLoadPart AND #i1s_Pulse) OR #iTest_Lamp;
END_REGION

REGION Network 5: 蜂鸣器蜂鸣次数 / Number of buzzer buzzes
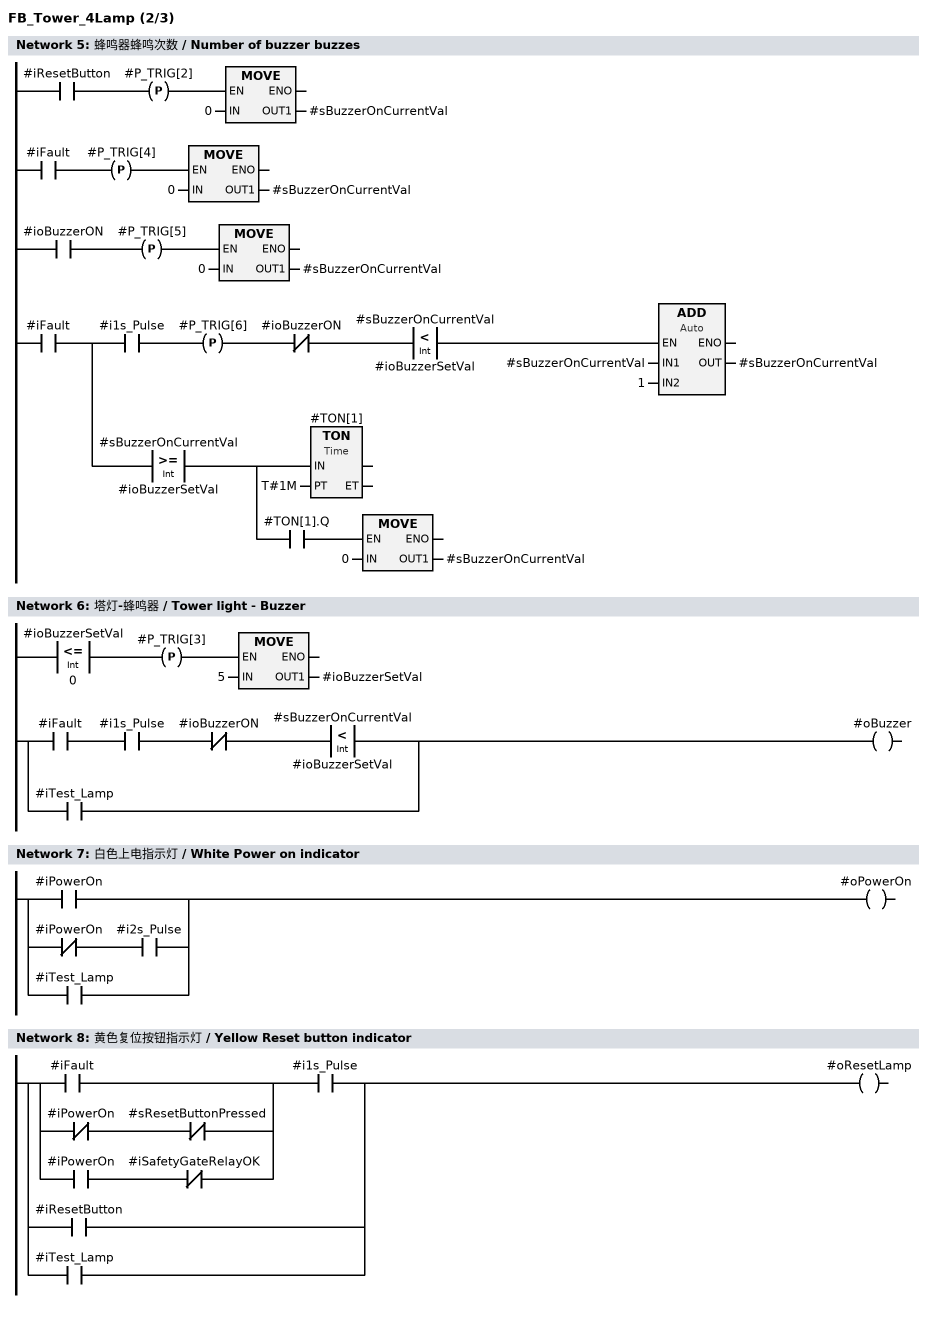
   RUNG wire#powerrail
      Contact( #iResetButton )
      P_Trig( #P_TRIG[2] )
      Move(in := 0, out1 => #sBuzzerOnCurrentVal)
   END_RUNG
   RUNG wire#powerrail
      Contact( #iFault )
      P_Trig( #P_TRIG[4] )
      Move(in := 0, out1 => #sBuzzerOnCurrentVal)
   END_RUNG
   RUNG wire#powerrail
      Contact( #ioBuzzerON )
      P_Trig( #P_TRIG[5] )
      Move(in := 0, out1 => #sBuzzerOnCurrentVal)
   END_RUNG
   RUNG wire#powerrail
      Contact( #iFault )
      wire#w1
      Contact( #i1s_Pulse )
      P_Trig( #P_TRIG[6] )
      I_Contact( #ioBuzzerON )
      { S7_Templates := "SrcType := Int" } LT_Contact(in1 := #sBuzzerOnCurrentVal, in2 := #ioBuzzerSetVal)
      Add(in1 := #sBuzzerOnCurrentVal, in2 := 1, out => #sBuzzerOnCurrentVal)
   END_RUNG
   RUNG wire#w1
      { S7_Templates := "SrcType := Int" } GE_Contact(in1 := #sBuzzerOnCurrentVal, in2 := #ioBuzzerSetVal)
      wire#w2
      { S7_Templates := "time_type := Time" } #TON[1].TON(pt := T#1M, et =>)
   END_RUNG
   RUNG wire#w2
      Contact( #TON[1].Q )
      Move(in := 0, out1 => #sBuzzerOnCurrentVal)
   END_RUNG
   // the same network as SCL:
   #_w1 := #iResetButton AND NOT #P_TRIG[2];   // rising edge
   #P_TRIG[2] := #iResetButton;
   IF #_w1 THEN #sBuzzerOnCurrentVal := 0; END_IF;
   #_w2 := #iFault AND NOT #P_TRIG[4];   // rising edge
   #P_TRIG[4] := #iFault;
   IF #_w2 THEN #sBuzzerOnCurrentVal := 0; END_IF;
   #_w3 := #ioBuzzerON AND NOT #P_TRIG[5];   // rising edge
   #P_TRIG[5] := #ioBuzzerON;
   IF #_w3 THEN #sBuzzerOnCurrentVal := 0; END_IF;
   #_w4 := #iFault AND #i1s_Pulse;
   #_w5 := #_w4 AND NOT #P_TRIG[6];   // rising edge
   #P_TRIG[6] := #_w4;
   IF #_w5 AND NOT #ioBuzzerON AND (#sBuzzerOnCurrentVal < #ioBuzzerSetVal) THEN
       #sBuzzerOnCurrentVal := #sBuzzerOnCurrentVal + 1;
   END_IF;
   #_w6 := #iFault AND (#sBuzzerOnCurrentVal >= #ioBuzzerSetVal);
   #TON[1].TON(IN := #_w6, PT := T#1M);
   IF #_w6 AND #TON[1].Q THEN #sBuzzerOnCurrentVal := 0; END_IF;
END_REGION

